    LOCAL PROC Path_Draw()
        MoveL point_0_clearance,v500,fine,GS25_ParallelGripper\WObj:=Workobject_1;
        MoveL point_0_contact,v500,fine,GS25_ParallelGripper\WObj:=Workobject_1;
        MoveL point_1_contact,v500,fine,GS25_ParallelGripper\WObj:=Workobject_1;
        MoveL point_1_clearance,v500,fine,GS25_ParallelGripper\WObj:=Workobject_1;
        MoveL point_2_clearance,v500,fine,GS25_ParallelGripper\WObj:=Workobject_1;
        MoveL point_2_contact,v500,fine,GS25_ParallelGripper\WObj:=Workobject_1;
        MoveL point_3_contact,v500,fine,GS25_ParallelGripper\WObj:=Workobject_1;
        MoveL point_3_clearance,v500,fine,GS25_ParallelGripper\WObj:=Workobject_1;
        MoveL point_4_clearance,v500,fine,GS25_ParallelGripper\WObj:=Workobject_1;
        MoveL point_4_contact,v500,fine,GS25_ParallelGripper\WObj:=Workobject_1;
        MoveL point_5_contact,v500,fine,GS25_ParallelGripper\WObj:=Workobject_1;
        MoveL point_5_clearance,v500,fine,GS25_ParallelGripper\WObj:=Workobject_1;
        MoveL point_6_clearance,v500,fine,GS25_ParallelGripper\WObj:=Workobject_1;
        MoveL point_6_contact,v500,fine,GS25_ParallelGripper\WObj:=Workobject_1;
        MoveL point_7_contact,v500,fine,GS25_ParallelGripper\WObj:=Workobject_1;
        MoveL point_7_clearance,v500,fine,GS25_ParallelGripper\WObj:=Workobject_1;
        MoveL point_8_clearance,v500,fine,GS25_ParallelGripper\WObj:=Workobject_1;
        MoveL point_8_contact,v500,fine,GS25_ParallelGripper\WObj:=Workobject_1;
        MoveL point_9_contact,v500,fine,GS25_ParallelGripper\WObj:=Workobject_1;
        MoveL point_9_clearance,v500,fine,GS25_ParallelGripper\WObj:=Workobject_1;
        MoveL point_10_clearance,v500,fine,GS25_ParallelGripper\WObj:=Workobject_1;
        MoveL point_10_contact,v500,fine,GS25_ParallelGripper\WObj:=Workobject_1;
        MoveL point_11_contact,v500,fine,GS25_ParallelGripper\WObj:=Workobject_1;
        MoveL point_11_clearance,v500,fine,GS25_ParallelGripper\WObj:=Workobject_1;
        MoveL point_12_clearance,v500,fine,GS25_ParallelGripper\WObj:=Workobject_1;
        MoveL point_12_contact,v500,fine,GS25_ParallelGripper\WObj:=Workobject_1;
        MoveL point_13_contact,v500,fine,GS25_ParallelGripper\WObj:=Workobject_1;
        MoveL point_13_clearance,v500,fine,GS25_ParallelGripper\WObj:=Workobject_1;
        MoveL point_14_clearance,v500,fine,GS25_ParallelGripper\WObj:=Workobject_1;
        MoveL point_14_contact,v500,fine,GS25_ParallelGripper\WObj:=Workobject_1;
        MoveL point_15_contact,v500,fine,GS25_ParallelGripper\WObj:=Workobject_1;
        MoveL point_15_clearance,v500,fine,GS25_ParallelGripper\WObj:=Workobject_1;
        MoveL point_16_clearance,v500,fine,GS25_ParallelGripper\WObj:=Workobject_1;
        MoveL point_16_contact,v500,fine,GS25_ParallelGripper\WObj:=Workobject_1;
        MoveL point_17_contact,v500,fine,GS25_ParallelGripper\WObj:=Workobject_1;
        MoveL point_17_clearance,v500,fine,GS25_ParallelGripper\WObj:=Workobject_1;
        MoveL point_18_clearance,v500,fine,GS25_ParallelGripper\WObj:=Workobject_1;
        MoveL point_18_contact,v500,fine,GS25_ParallelGripper\WObj:=Workobject_1;
        MoveL point_19_contact,v500,fine,GS25_ParallelGripper\WObj:=Workobject_1;
        MoveL point_19_clearance,v500,fine,GS25_ParallelGripper\WObj:=Workobject_1;
        MoveL point_20_clearance,v500,fine,GS25_ParallelGripper\WObj:=Workobject_1;
        MoveL point_20_contact,v500,fine,GS25_ParallelGripper\WObj:=Workobject_1;
        MoveL point_21_contact,v500,fine,GS25_ParallelGripper\WObj:=Workobject_1;
        MoveL point_21_clearance,v500,fine,GS25_ParallelGripper\WObj:=Workobject_1;
        MoveL point_22_clearance,v500,fine,GS25_ParallelGripper\WObj:=Workobject_1;
        MoveL point_22_contact,v500,fine,GS25_ParallelGripper\WObj:=Workobject_1;
        MoveL point_23_contact,v500,fine,GS25_ParallelGripper\WObj:=Workobject_1;
        MoveL point_23_clearance,v500,fine,GS25_ParallelGripper\WObj:=Workobject_1;
        MoveL point_24_clearance,v500,fine,GS25_ParallelGripper\WObj:=Workobject_1;
        MoveL point_24_contact,v500,fine,GS25_ParallelGripper\WObj:=Workobject_1;
        MoveL point_25_contact,v500,fine,GS25_ParallelGripper\WObj:=Workobject_1;
        MoveL point_25_clearance,v500,fine,GS25_ParallelGripper\WObj:=Workobject_1;
        MoveL point_26_clearance,v500,fine,GS25_ParallelGripper\WObj:=Workobject_1;
        MoveL point_26_contact,v500,fine,GS25_ParallelGripper\WObj:=Workobject_1;
        MoveL point_27_contact,v500,fine,GS25_ParallelGripper\WObj:=Workobject_1;
        MoveL point_27_clearance,v500,fine,GS25_ParallelGripper\WObj:=Workobject_1;
        MoveL point_28_clearance,v500,fine,GS25_ParallelGripper\WObj:=Workobject_1;
        MoveL point_28_contact,v500,fine,GS25_ParallelGripper\WObj:=Workobject_1;
        MoveL point_29_contact,v500,fine,GS25_ParallelGripper\WObj:=Workobject_1;
        MoveL point_29_clearance,v500,fine,GS25_ParallelGripper\WObj:=Workobject_1;
        MoveL point_30_clearance,v500,fine,GS25_ParallelGripper\WObj:=Workobject_1;
        MoveL point_30_contact,v500,fine,GS25_ParallelGripper\WObj:=Workobject_1;
        MoveL point_31_contact,v500,fine,GS25_ParallelGripper\WObj:=Workobject_1;
        MoveL point_31_clearance,v500,fine,GS25_ParallelGripper\WObj:=Workobject_1;
        MoveL point_32_clearance,v500,fine,GS25_ParallelGripper\WObj:=Workobject_1;
        MoveL point_32_contact,v500,fine,GS25_ParallelGripper\WObj:=Workobject_1;
        MoveL point_33_contact,v500,fine,GS25_ParallelGripper\WObj:=Workobject_1;
        MoveL point_33_clearance,v500,fine,GS25_ParallelGripper\WObj:=Workobject_1;
        MoveL point_34_clearance,v500,fine,GS25_ParallelGripper\WObj:=Workobject_1;
        MoveL point_34_contact,v500,fine,GS25_ParallelGripper\WObj:=Workobject_1;
        MoveL point_35_contact,v500,fine,GS25_ParallelGripper\WObj:=Workobject_1;
        MoveL point_35_clearance,v500,fine,GS25_ParallelGripper\WObj:=Workobject_1;
        MoveL point_36_clearance,v500,fine,GS25_ParallelGripper\WObj:=Workobject_1;
        MoveL point_36_contact,v500,fine,GS25_ParallelGripper\WObj:=Workobject_1;
        MoveL point_37_contact,v500,fine,GS25_ParallelGripper\WObj:=Workobject_1;
        MoveL point_37_clearance,v500,fine,GS25_ParallelGripper\WObj:=Workobject_1;
        MoveL point_38_clearance,v500,fine,GS25_ParallelGripper\WObj:=Workobject_1;
        MoveL point_38_contact,v500,fine,GS25_ParallelGripper\WObj:=Workobject_1;
        MoveL point_39_contact,v500,fine,GS25_ParallelGripper\WObj:=Workobject_1;
        MoveL point_39_clearance,v500,fine,GS25_ParallelGripper\WObj:=Workobject_1;
        MoveL point_40_clearance,v500,fine,GS25_ParallelGripper\WObj:=Workobject_1;
        MoveL point_40_contact,v500,fine,GS25_ParallelGripper\WObj:=Workobject_1;
        MoveL point_41_contact,v500,fine,GS25_ParallelGripper\WObj:=Workobject_1;
        MoveL point_41_clearance,v500,fine,GS25_ParallelGripper\WObj:=Workobject_1;
        MoveL point_42_clearance,v500,fine,GS25_ParallelGripper\WObj:=Workobject_1;
        MoveL point_42_contact,v500,fine,GS25_ParallelGripper\WObj:=Workobject_1;
        MoveL point_43_contact,v500,fine,GS25_ParallelGripper\WObj:=Workobject_1;
        MoveL point_43_clearance,v500,fine,GS25_ParallelGripper\WObj:=Workobject_1;
        MoveL point_44_clearance,v500,fine,GS25_ParallelGripper\WObj:=Workobject_1;
        MoveL point_44_contact,v500,fine,GS25_ParallelGripper\WObj:=Workobject_1;
        MoveL point_45_contact,v500,fine,GS25_ParallelGripper\WObj:=Workobject_1;
        MoveL point_45_clearance,v500,fine,GS25_ParallelGripper\WObj:=Workobject_1;
        MoveL point_46_clearance,v500,fine,GS25_ParallelGripper\WObj:=Workobject_1;
        MoveL point_46_contact,v500,fine,GS25_ParallelGripper\WObj:=Workobject_1;
        MoveL point_47_contact,v500,fine,GS25_ParallelGripper\WObj:=Workobject_1;
        MoveL point_47_clearance,v500,fine,GS25_ParallelGripper\WObj:=Workobject_1;
        MoveL point_48_clearance,v500,fine,GS25_ParallelGripper\WObj:=Workobject_1;
        MoveL point_48_contact,v500,fine,GS25_ParallelGripper\WObj:=Workobject_1;
        MoveL point_49_contact,v500,fine,GS25_ParallelGripper\WObj:=Workobject_1;
        MoveL point_49_clearance,v500,fine,GS25_ParallelGripper\WObj:=Workobject_1;
        MoveL point_50_clearance,v500,fine,GS25_ParallelGripper\WObj:=Workobject_1;
        MoveL point_50_contact,v500,fine,GS25_ParallelGripper\WObj:=Workobject_1;
        MoveL point_51_contact,v500,fine,GS25_ParallelGripper\WObj:=Workobject_1;
        MoveL point_51_clearance,v500,fine,GS25_ParallelGripper\WObj:=Workobject_1;
        MoveL point_52_clearance,v500,fine,GS25_ParallelGripper\WObj:=Workobject_1;
        MoveL point_52_contact,v500,fine,GS25_ParallelGripper\WObj:=Workobject_1;
        MoveL point_53_contact,v500,fine,GS25_ParallelGripper\WObj:=Workobject_1;
        MoveL point_53_clearance,v500,fine,GS25_ParallelGripper\WObj:=Workobject_1;
        MoveL point_54_clearance,v500,fine,GS25_ParallelGripper\WObj:=Workobject_1;
        MoveL point_54_contact,v500,fine,GS25_ParallelGripper\WObj:=Workobject_1;
        MoveL point_55_contact,v500,fine,GS25_ParallelGripper\WObj:=Workobject_1;
        MoveL point_55_clearance,v500,fine,GS25_ParallelGripper\WObj:=Workobject_1;
        MoveL point_56_clearance,v500,fine,GS25_ParallelGripper\WObj:=Workobject_1;
        MoveL point_56_contact,v500,fine,GS25_ParallelGripper\WObj:=Workobject_1;
        MoveL point_57_contact,v500,fine,GS25_ParallelGripper\WObj:=Workobject_1;
        MoveL point_57_clearance,v500,fine,GS25_ParallelGripper\WObj:=Workobject_1;
        MoveL point_58_clearance,v500,fine,GS25_ParallelGripper\WObj:=Workobject_1;
        MoveL point_58_contact,v500,fine,GS25_ParallelGripper\WObj:=Workobject_1;
        MoveL point_59_contact,v500,fine,GS25_ParallelGripper\WObj:=Workobject_1;
        MoveL point_59_clearance,v500,fine,GS25_ParallelGripper\WObj:=Workobject_1;
        MoveL point_60_clearance,v500,fine,GS25_ParallelGripper\WObj:=Workobject_1;
        MoveL point_60_contact,v500,fine,GS25_ParallelGripper\WObj:=Workobject_1;
        MoveL point_61_contact,v500,fine,GS25_ParallelGripper\WObj:=Workobject_1;
        MoveL point_61_clearance,v500,fine,GS25_ParallelGripper\WObj:=Workobject_1;
        MoveL point_62_clearance,v500,fine,GS25_ParallelGripper\WObj:=Workobject_1;
        MoveL point_62_contact,v500,fine,GS25_ParallelGripper\WObj:=Workobject_1;
        MoveL point_63_contact,v500,fine,GS25_ParallelGripper\WObj:=Workobject_1;
        MoveL point_63_clearance,v500,fine,GS25_ParallelGripper\WObj:=Workobject_1;
        MoveL point_64_clearance,v500,fine,GS25_ParallelGripper\WObj:=Workobject_1;
        MoveL point_64_contact,v500,fine,GS25_ParallelGripper\WObj:=Workobject_1;
        MoveL point_65_contact,v500,fine,GS25_ParallelGripper\WObj:=Workobject_1;
        MoveL point_65_clearance,v500,fine,GS25_ParallelGripper\WObj:=Workobject_1;
        MoveL point_66_clearance,v500,fine,GS25_ParallelGripper\WObj:=Workobject_1;
        MoveL point_66_contact,v500,fine,GS25_ParallelGripper\WObj:=Workobject_1;
        MoveL point_67_contact,v500,fine,GS25_ParallelGripper\WObj:=Workobject_1;
        MoveL point_67_clearance,v500,fine,GS25_ParallelGripper\WObj:=Workobject_1;
        MoveL point_68_clearance,v500,fine,GS25_ParallelGripper\WObj:=Workobject_1;
        MoveL point_68_contact,v500,fine,GS25_ParallelGripper\WObj:=Workobject_1;
        MoveL point_69_contact,v500,fine,GS25_ParallelGripper\WObj:=Workobject_1;
        MoveL point_69_clearance,v500,fine,GS25_ParallelGripper\WObj:=Workobject_1;
        MoveL point_70_clearance,v500,fine,GS25_ParallelGripper\WObj:=Workobject_1;
        MoveL point_70_contact,v500,fine,GS25_ParallelGripper\WObj:=Workobject_1;
        MoveL point_71_contact,v500,fine,GS25_ParallelGripper\WObj:=Workobject_1;
        MoveL point_71_clearance,v500,fine,GS25_ParallelGripper\WObj:=Workobject_1;
        MoveL point_72_clearance,v500,fine,GS25_ParallelGripper\WObj:=Workobject_1;
        MoveL point_72_contact,v500,fine,GS25_ParallelGripper\WObj:=Workobject_1;
        MoveL point_73_contact,v500,fine,GS25_ParallelGripper\WObj:=Workobject_1;
        MoveL point_73_clearance,v500,fine,GS25_ParallelGripper\WObj:=Workobject_1;
        MoveL point_74_clearance,v500,fine,GS25_ParallelGripper\WObj:=Workobject_1;
        MoveL point_74_contact,v500,fine,GS25_ParallelGripper\WObj:=Workobject_1;
        MoveL point_75_contact,v500,fine,GS25_ParallelGripper\WObj:=Workobject_1;
        MoveL point_75_clearance,v500,fine,GS25_ParallelGripper\WObj:=Workobject_1;
        MoveL point_76_clearance,v500,fine,GS25_ParallelGripper\WObj:=Workobject_1;
        MoveL point_76_contact,v500,fine,GS25_ParallelGripper\WObj:=Workobject_1;
        MoveL point_77_contact,v500,fine,GS25_ParallelGripper\WObj:=Workobject_1;
        MoveL point_77_clearance,v500,fine,GS25_ParallelGripper\WObj:=Workobject_1;
        MoveL point_78_clearance,v500,fine,GS25_ParallelGripper\WObj:=Workobject_1;
        MoveL point_78_contact,v500,fine,GS25_ParallelGripper\WObj:=Workobject_1;
        MoveL point_79_contact,v500,fine,GS25_ParallelGripper\WObj:=Workobject_1;
        MoveL point_79_clearance,v500,fine,GS25_ParallelGripper\WObj:=Workobject_1;
        MoveL point_80_clearance,v500,fine,GS25_ParallelGripper\WObj:=Workobject_1;
        MoveL point_80_contact,v500,fine,GS25_ParallelGripper\WObj:=Workobject_1;
        MoveL point_81_contact,v500,fine,GS25_ParallelGripper\WObj:=Workobject_1;
        MoveL point_81_clearance,v500,fine,GS25_ParallelGripper\WObj:=Workobject_1;
        MoveL point_82_clearance,v500,fine,GS25_ParallelGripper\WObj:=Workobject_1;
        MoveL point_82_contact,v500,fine,GS25_ParallelGripper\WObj:=Workobject_1;
        MoveL point_83_contact,v500,fine,GS25_ParallelGripper\WObj:=Workobject_1;
        MoveL point_83_clearance,v500,fine,GS25_ParallelGripper\WObj:=Workobject_1;
        MoveL point_84_clearance,v500,fine,GS25_ParallelGripper\WObj:=Workobject_1;
        MoveL point_84_contact,v500,fine,GS25_ParallelGripper\WObj:=Workobject_1;
        MoveL point_85_contact,v500,fine,GS25_ParallelGripper\WObj:=Workobject_1;
        MoveL point_85_clearance,v500,fine,GS25_ParallelGripper\WObj:=Workobject_1;
        MoveL point_86_clearance,v500,fine,GS25_ParallelGripper\WObj:=Workobject_1;
        MoveL point_86_contact,v500,fine,GS25_ParallelGripper\WObj:=Workobject_1;
        MoveL point_87_contact,v500,fine,GS25_ParallelGripper\WObj:=Workobject_1;
        MoveL point_87_clearance,v500,fine,GS25_ParallelGripper\WObj:=Workobject_1;
        MoveL point_88_clearance,v500,fine,GS25_ParallelGripper\WObj:=Workobject_1;
        MoveL point_88_contact,v500,fine,GS25_ParallelGripper\WObj:=Workobject_1;
        MoveL point_89_contact,v500,fine,GS25_ParallelGripper\WObj:=Workobject_1;
        MoveL point_89_clearance,v500,fine,GS25_ParallelGripper\WObj:=Workobject_1;
        MoveL point_90_clearance,v500,fine,GS25_ParallelGripper\WObj:=Workobject_1;
        MoveL point_90_contact,v500,fine,GS25_ParallelGripper\WObj:=Workobject_1;
        MoveL point_91_contact,v500,fine,GS25_ParallelGripper\WObj:=Workobject_1;
        MoveL point_91_clearance,v500,fine,GS25_ParallelGripper\WObj:=Workobject_1;
        MoveL point_92_clearance,v500,fine,GS25_ParallelGripper\WObj:=Workobject_1;
        MoveL point_92_contact,v500,fine,GS25_ParallelGripper\WObj:=Workobject_1;
        MoveL point_93_contact,v500,fine,GS25_ParallelGripper\WObj:=Workobject_1;
        MoveL point_93_clearance,v500,fine,GS25_ParallelGripper\WObj:=Workobject_1;
        MoveL point_94_clearance,v500,fine,GS25_ParallelGripper\WObj:=Workobject_1;
        MoveL point_94_contact,v500,fine,GS25_ParallelGripper\WObj:=Workobject_1;
        MoveL point_95_contact,v500,fine,GS25_ParallelGripper\WObj:=Workobject_1;
        MoveL point_95_clearance,v500,fine,GS25_ParallelGripper\WObj:=Workobject_1;
        MoveL point_96_clearance,v500,fine,GS25_ParallelGripper\WObj:=Workobject_1;
        MoveL point_96_contact,v500,fine,GS25_ParallelGripper\WObj:=Workobject_1;
        MoveL point_97_contact,v500,fine,GS25_ParallelGripper\WObj:=Workobject_1;
        MoveL point_97_clearance,v500,fine,GS25_ParallelGripper\WObj:=Workobject_1;
        MoveL point_98_clearance,v500,fine,GS25_ParallelGripper\WObj:=Workobject_1;
        MoveL point_98_contact,v500,fine,GS25_ParallelGripper\WObj:=Workobject_1;
        MoveL point_99_contact,v500,fine,GS25_ParallelGripper\WObj:=Workobject_1;
        MoveL point_99_clearance,v500,fine,GS25_ParallelGripper\WObj:=Workobject_1;
        MoveL point_100_clearance,v500,fine,GS25_ParallelGripper\WObj:=Workobject_1;
        MoveL point_100_contact,v500,fine,GS25_ParallelGripper\WObj:=Workobject_1;
        MoveL point_101_contact,v500,fine,GS25_ParallelGripper\WObj:=Workobject_1;
        MoveL point_101_clearance,v500,fine,GS25_ParallelGripper\WObj:=Workobject_1;
        MoveL point_102_clearance,v500,fine,GS25_ParallelGripper\WObj:=Workobject_1;
        MoveL point_102_contact,v500,fine,GS25_ParallelGripper\WObj:=Workobject_1;
        MoveL point_103_contact,v500,fine,GS25_ParallelGripper\WObj:=Workobject_1;
        MoveL point_103_clearance,v500,fine,GS25_ParallelGripper\WObj:=Workobject_1;
        MoveL point_104_clearance,v500,fine,GS25_ParallelGripper\WObj:=Workobject_1;
        MoveL point_104_contact,v500,fine,GS25_ParallelGripper\WObj:=Workobject_1;
        MoveL point_105_contact,v500,fine,GS25_ParallelGripper\WObj:=Workobject_1;
        MoveL point_105_clearance,v500,fine,GS25_ParallelGripper\WObj:=Workobject_1;
        MoveL point_106_clearance,v500,fine,GS25_ParallelGripper\WObj:=Workobject_1;
        MoveL point_106_contact,v500,fine,GS25_ParallelGripper\WObj:=Workobject_1;
        MoveL point_107_contact,v500,fine,GS25_ParallelGripper\WObj:=Workobject_1;
        MoveL point_107_clearance,v500,fine,GS25_ParallelGripper\WObj:=Workobject_1;
        MoveL point_108_clearance,v500,fine,GS25_ParallelGripper\WObj:=Workobject_1;
        MoveL point_108_contact,v500,fine,GS25_ParallelGripper\WObj:=Workobject_1;
        MoveL point_109_contact,v500,fine,GS25_ParallelGripper\WObj:=Workobject_1;
        MoveL point_109_clearance,v500,fine,GS25_ParallelGripper\WObj:=Workobject_1;
        MoveL point_110_clearance,v500,fine,GS25_ParallelGripper\WObj:=Workobject_1;
        MoveL point_110_contact,v500,fine,GS25_ParallelGripper\WObj:=Workobject_1;
        MoveL point_111_contact,v500,fine,GS25_ParallelGripper\WObj:=Workobject_1;
        MoveL point_111_clearance,v500,fine,GS25_ParallelGripper\WObj:=Workobject_1;
        MoveL point_112_clearance,v500,fine,GS25_ParallelGripper\WObj:=Workobject_1;
        MoveL point_112_contact,v500,fine,GS25_ParallelGripper\WObj:=Workobject_1;
        MoveL point_113_contact,v500,fine,GS25_ParallelGripper\WObj:=Workobject_1;
        MoveL point_113_clearance,v500,fine,GS25_ParallelGripper\WObj:=Workobject_1;
        MoveL point_114_clearance,v500,fine,GS25_ParallelGripper\WObj:=Workobject_1;
        MoveL point_114_contact,v500,fine,GS25_ParallelGripper\WObj:=Workobject_1;
        MoveL point_115_contact,v500,fine,GS25_ParallelGripper\WObj:=Workobject_1;
        MoveL point_115_clearance,v500,fine,GS25_ParallelGripper\WObj:=Workobject_1;
        MoveL point_116_clearance,v500,fine,GS25_ParallelGripper\WObj:=Workobject_1;
        MoveL point_116_contact,v500,fine,GS25_ParallelGripper\WObj:=Workobject_1;
        MoveL point_117_contact,v500,fine,GS25_ParallelGripper\WObj:=Workobject_1;
        MoveL point_117_clearance,v500,fine,GS25_ParallelGripper\WObj:=Workobject_1;
        MoveL point_118_clearance,v500,fine,GS25_ParallelGripper\WObj:=Workobject_1;
        MoveL point_118_contact,v500,fine,GS25_ParallelGripper\WObj:=Workobject_1;
        MoveL point_119_contact,v500,fine,GS25_ParallelGripper\WObj:=Workobject_1;
        MoveL point_119_clearance,v500,fine,GS25_ParallelGripper\WObj:=Workobject_1;
        MoveL point_120_clearance,v500,fine,GS25_ParallelGripper\WObj:=Workobject_1;
        MoveL point_120_contact,v500,fine,GS25_ParallelGripper\WObj:=Workobject_1;
        MoveL point_121_contact,v500,fine,GS25_ParallelGripper\WObj:=Workobject_1;
        MoveL point_121_clearance,v500,fine,GS25_ParallelGripper\WObj:=Workobject_1;
        MoveL point_122_clearance,v500,fine,GS25_ParallelGripper\WObj:=Workobject_1;
        MoveL point_122_contact,v500,fine,GS25_ParallelGripper\WObj:=Workobject_1;
        MoveL point_123_contact,v500,fine,GS25_ParallelGripper\WObj:=Workobject_1;
        MoveL point_123_clearance,v500,fine,GS25_ParallelGripper\WObj:=Workobject_1;
        MoveL point_124_clearance,v500,fine,GS25_ParallelGripper\WObj:=Workobject_1;
        MoveL point_124_contact,v500,fine,GS25_ParallelGripper\WObj:=Workobject_1;
        MoveL point_125_contact,v500,fine,GS25_ParallelGripper\WObj:=Workobject_1;
        MoveL point_125_clearance,v500,fine,GS25_ParallelGripper\WObj:=Workobject_1;
        MoveL point_126_clearance,v500,fine,GS25_ParallelGripper\WObj:=Workobject_1;
        MoveL point_126_contact,v500,fine,GS25_ParallelGripper\WObj:=Workobject_1;
        MoveL point_127_contact,v500,fine,GS25_ParallelGripper\WObj:=Workobject_1;
        MoveL point_127_clearance,v500,fine,GS25_ParallelGripper\WObj:=Workobject_1;
        MoveL point_128_clearance,v500,fine,GS25_ParallelGripper\WObj:=Workobject_1;
        MoveL point_128_contact,v500,fine,GS25_ParallelGripper\WObj:=Workobject_1;
        MoveL point_129_contact,v500,fine,GS25_ParallelGripper\WObj:=Workobject_1;
        MoveL point_129_clearance,v500,fine,GS25_ParallelGripper\WObj:=Workobject_1;
        MoveL point_130_clearance,v500,fine,GS25_ParallelGripper\WObj:=Workobject_1;
        MoveL point_130_contact,v500,fine,GS25_ParallelGripper\WObj:=Workobject_1;
        MoveL point_131_contact,v500,fine,GS25_ParallelGripper\WObj:=Workobject_1;
        MoveL point_131_clearance,v500,fine,GS25_ParallelGripper\WObj:=Workobject_1;
        MoveL point_132_clearance,v500,fine,GS25_ParallelGripper\WObj:=Workobject_1;
        MoveL point_132_contact,v500,fine,GS25_ParallelGripper\WObj:=Workobject_1;
        MoveL point_133_contact,v500,fine,GS25_ParallelGripper\WObj:=Workobject_1;
        MoveL point_133_clearance,v500,fine,GS25_ParallelGripper\WObj:=Workobject_1;
        MoveL point_134_clearance,v500,fine,GS25_ParallelGripper\WObj:=Workobject_1;
        MoveL point_134_contact,v500,fine,GS25_ParallelGripper\WObj:=Workobject_1;
        MoveL point_135_contact,v500,fine,GS25_ParallelGripper\WObj:=Workobject_1;
        MoveL point_135_clearance,v500,fine,GS25_ParallelGripper\WObj:=Workobject_1;
        MoveL point_136_clearance,v500,fine,GS25_ParallelGripper\WObj:=Workobject_1;
        MoveL point_136_contact,v500,fine,GS25_ParallelGripper\WObj:=Workobject_1;
        MoveL point_137_contact,v500,fine,GS25_ParallelGripper\WObj:=Workobject_1;
        MoveL point_137_clearance,v500,fine,GS25_ParallelGripper\WObj:=Workobject_1;
        MoveL point_138_clearance,v500,fine,GS25_ParallelGripper\WObj:=Workobject_1;
        MoveL point_138_contact,v500,fine,GS25_ParallelGripper\WObj:=Workobject_1;
        MoveL point_139_contact,v500,fine,GS25_ParallelGripper\WObj:=Workobject_1;
        MoveL point_139_clearance,v500,fine,GS25_ParallelGripper\WObj:=Workobject_1;
        MoveL point_140_clearance,v500,fine,GS25_ParallelGripper\WObj:=Workobject_1;
        MoveL point_140_contact,v500,fine,GS25_ParallelGripper\WObj:=Workobject_1;
        MoveL point_141_contact,v500,fine,GS25_ParallelGripper\WObj:=Workobject_1;
        MoveL point_141_clearance,v500,fine,GS25_ParallelGripper\WObj:=Workobject_1;
        MoveL point_142_clearance,v500,fine,GS25_ParallelGripper\WObj:=Workobject_1;
        MoveL point_142_contact,v500,fine,GS25_ParallelGripper\WObj:=Workobject_1;
        MoveL point_143_contact,v500,fine,GS25_ParallelGripper\WObj:=Workobject_1;
        MoveL point_143_clearance,v500,fine,GS25_ParallelGripper\WObj:=Workobject_1;
        MoveL point_144_clearance,v500,fine,GS25_ParallelGripper\WObj:=Workobject_1;
        MoveL point_144_contact,v500,fine,GS25_ParallelGripper\WObj:=Workobject_1;
        MoveL point_145_contact,v500,fine,GS25_ParallelGripper\WObj:=Workobject_1;
        MoveL point_145_clearance,v500,fine,GS25_ParallelGripper\WObj:=Workobject_1;
        MoveL point_146_clearance,v500,fine,GS25_ParallelGripper\WObj:=Workobject_1;
        MoveL point_146_contact,v500,fine,GS25_ParallelGripper\WObj:=Workobject_1;
        MoveL point_147_contact,v500,fine,GS25_ParallelGripper\WObj:=Workobject_1;
        MoveL point_147_clearance,v500,fine,GS25_ParallelGripper\WObj:=Workobject_1;
        MoveL point_148_clearance,v500,fine,GS25_ParallelGripper\WObj:=Workobject_1;
        MoveL point_148_contact,v500,fine,GS25_ParallelGripper\WObj:=Workobject_1;
        MoveL point_149_contact,v500,fine,GS25_ParallelGripper\WObj:=Workobject_1;
        MoveL point_149_clearance,v500,fine,GS25_ParallelGripper\WObj:=Workobject_1;
        MoveL point_150_clearance,v500,fine,GS25_ParallelGripper\WObj:=Workobject_1;
        MoveL point_150_contact,v500,fine,GS25_ParallelGripper\WObj:=Workobject_1;
        MoveL point_151_contact,v500,fine,GS25_ParallelGripper\WObj:=Workobject_1;
        MoveL point_151_clearance,v500,fine,GS25_ParallelGripper\WObj:=Workobject_1;
        MoveL point_152_clearance,v500,fine,GS25_ParallelGripper\WObj:=Workobject_1;
        MoveL point_152_contact,v500,fine,GS25_ParallelGripper\WObj:=Workobject_1;
        MoveL point_153_contact,v500,fine,GS25_ParallelGripper\WObj:=Workobject_1;
        MoveL point_153_clearance,v500,fine,GS25_ParallelGripper\WObj:=Workobject_1;
        MoveL point_154_clearance,v500,fine,GS25_ParallelGripper\WObj:=Workobject_1;
        MoveL point_154_contact,v500,fine,GS25_ParallelGripper\WObj:=Workobject_1;
        MoveL point_155_contact,v500,fine,GS25_ParallelGripper\WObj:=Workobject_1;
        MoveL point_155_clearance,v500,fine,GS25_ParallelGripper\WObj:=Workobject_1;
        MoveL point_156_clearance,v500,fine,GS25_ParallelGripper\WObj:=Workobject_1;
        MoveL point_156_contact,v500,fine,GS25_ParallelGripper\WObj:=Workobject_1;
        MoveL point_157_contact,v500,fine,GS25_ParallelGripper\WObj:=Workobject_1;
        MoveL point_157_clearance,v500,fine,GS25_ParallelGripper\WObj:=Workobject_1;
        MoveL point_158_clearance,v500,fine,GS25_ParallelGripper\WObj:=Workobject_1;
        MoveL point_158_contact,v500,fine,GS25_ParallelGripper\WObj:=Workobject_1;
        MoveL point_159_contact,v500,fine,GS25_ParallelGripper\WObj:=Workobject_1;
        MoveL point_159_clearance,v500,fine,GS25_ParallelGripper\WObj:=Workobject_1;
        MoveL point_160_clearance,v500,fine,GS25_ParallelGripper\WObj:=Workobject_1;
        MoveL point_160_contact,v500,fine,GS25_ParallelGripper\WObj:=Workobject_1;
        MoveL point_161_contact,v500,fine,GS25_ParallelGripper\WObj:=Workobject_1;
        MoveL point_161_clearance,v500,fine,GS25_ParallelGripper\WObj:=Workobject_1;
        MoveL point_162_clearance,v500,fine,GS25_ParallelGripper\WObj:=Workobject_1;
        MoveL point_162_contact,v500,fine,GS25_ParallelGripper\WObj:=Workobject_1;
        MoveL point_163_contact,v500,fine,GS25_ParallelGripper\WObj:=Workobject_1;
        MoveL point_163_clearance,v500,fine,GS25_ParallelGripper\WObj:=Workobject_1;
        MoveL point_164_clearance,v500,fine,GS25_ParallelGripper\WObj:=Workobject_1;
        MoveL point_164_contact,v500,fine,GS25_ParallelGripper\WObj:=Workobject_1;
        MoveL point_165_contact,v500,fine,GS25_ParallelGripper\WObj:=Workobject_1;
        MoveL point_165_clearance,v500,fine,GS25_ParallelGripper\WObj:=Workobject_1;
        MoveL point_166_clearance,v500,fine,GS25_ParallelGripper\WObj:=Workobject_1;
        MoveL point_166_contact,v500,fine,GS25_ParallelGripper\WObj:=Workobject_1;
        MoveL point_167_contact,v500,fine,GS25_ParallelGripper\WObj:=Workobject_1;
        MoveL point_167_clearance,v500,fine,GS25_ParallelGripper\WObj:=Workobject_1;
        MoveL point_168_clearance,v500,fine,GS25_ParallelGripper\WObj:=Workobject_1;
        MoveL point_168_contact,v500,fine,GS25_ParallelGripper\WObj:=Workobject_1;
        MoveL point_169_contact,v500,fine,GS25_ParallelGripper\WObj:=Workobject_1;
        MoveL point_169_clearance,v500,fine,GS25_ParallelGripper\WObj:=Workobject_1;
        MoveL point_170_clearance,v500,fine,GS25_ParallelGripper\WObj:=Workobject_1;
        MoveL point_170_contact,v500,fine,GS25_ParallelGripper\WObj:=Workobject_1;
        MoveL point_171_contact,v500,fine,GS25_ParallelGripper\WObj:=Workobject_1;
        MoveL point_171_clearance,v500,fine,GS25_ParallelGripper\WObj:=Workobject_1;
        MoveL point_172_clearance,v500,fine,GS25_ParallelGripper\WObj:=Workobject_1;
        MoveL point_172_contact,v500,fine,GS25_ParallelGripper\WObj:=Workobject_1;
        MoveL point_173_contact,v500,fine,GS25_ParallelGripper\WObj:=Workobject_1;
        MoveL point_173_clearance,v500,fine,GS25_ParallelGripper\WObj:=Workobject_1;
        MoveL point_174_clearance,v500,fine,GS25_ParallelGripper\WObj:=Workobject_1;
        MoveL point_174_contact,v500,fine,GS25_ParallelGripper\WObj:=Workobject_1;
        MoveL point_175_contact,v500,fine,GS25_ParallelGripper\WObj:=Workobject_1;
        MoveL point_175_clearance,v500,fine,GS25_ParallelGripper\WObj:=Workobject_1;
        MoveL point_176_clearance,v500,fine,GS25_ParallelGripper\WObj:=Workobject_1;
        MoveL point_176_contact,v500,fine,GS25_ParallelGripper\WObj:=Workobject_1;
        MoveL point_177_contact,v500,fine,GS25_ParallelGripper\WObj:=Workobject_1;
        MoveL point_177_clearance,v500,fine,GS25_ParallelGripper\WObj:=Workobject_1;
        MoveL point_178_clearance,v500,fine,GS25_ParallelGripper\WObj:=Workobject_1;
        MoveL point_178_contact,v500,fine,GS25_ParallelGripper\WObj:=Workobject_1;
        MoveL point_179_contact,v500,fine,GS25_ParallelGripper\WObj:=Workobject_1;
        MoveL point_179_clearance,v500,fine,GS25_ParallelGripper\WObj:=Workobject_1;
        MoveL point_180_clearance,v500,fine,GS25_ParallelGripper\WObj:=Workobject_1;
        MoveL point_180_contact,v500,fine,GS25_ParallelGripper\WObj:=Workobject_1;
        MoveL point_181_contact,v500,fine,GS25_ParallelGripper\WObj:=Workobject_1;
        MoveL point_181_clearance,v500,fine,GS25_ParallelGripper\WObj:=Workobject_1;
        MoveL point_182_clearance,v500,fine,GS25_ParallelGripper\WObj:=Workobject_1;
        MoveL point_182_contact,v500,fine,GS25_ParallelGripper\WObj:=Workobject_1;
        MoveL point_183_contact,v500,fine,GS25_ParallelGripper\WObj:=Workobject_1;
        MoveL point_183_clearance,v500,fine,GS25_ParallelGripper\WObj:=Workobject_1;
        MoveL point_184_clearance,v500,fine,GS25_ParallelGripper\WObj:=Workobject_1;
        MoveL point_184_contact,v500,fine,GS25_ParallelGripper\WObj:=Workobject_1;
        MoveL point_185_contact,v500,fine,GS25_ParallelGripper\WObj:=Workobject_1;
        MoveL point_185_clearance,v500,fine,GS25_ParallelGripper\WObj:=Workobject_1;
        MoveL point_186_clearance,v500,fine,GS25_ParallelGripper\WObj:=Workobject_1;
        MoveL point_186_contact,v500,fine,GS25_ParallelGripper\WObj:=Workobject_1;
        MoveL point_187_contact,v500,fine,GS25_ParallelGripper\WObj:=Workobject_1;
        MoveL point_187_clearance,v500,fine,GS25_ParallelGripper\WObj:=Workobject_1;
        MoveL point_188_clearance,v500,fine,GS25_ParallelGripper\WObj:=Workobject_1;
        MoveL point_188_contact,v500,fine,GS25_ParallelGripper\WObj:=Workobject_1;
        MoveL point_189_contact,v500,fine,GS25_ParallelGripper\WObj:=Workobject_1;
        MoveL point_189_clearance,v500,fine,GS25_ParallelGripper\WObj:=Workobject_1;
        MoveL point_190_clearance,v500,fine,GS25_ParallelGripper\WObj:=Workobject_1;
        MoveL point_190_contact,v500,fine,GS25_ParallelGripper\WObj:=Workobject_1;
        MoveL point_191_contact,v500,fine,GS25_ParallelGripper\WObj:=Workobject_1;
        MoveL point_191_clearance,v500,fine,GS25_ParallelGripper\WObj:=Workobject_1;
        MoveL point_192_clearance,v500,fine,GS25_ParallelGripper\WObj:=Workobject_1;
        MoveL point_192_contact,v500,fine,GS25_ParallelGripper\WObj:=Workobject_1;
        MoveL point_193_contact,v500,fine,GS25_ParallelGripper\WObj:=Workobject_1;
        MoveL point_193_clearance,v500,fine,GS25_ParallelGripper\WObj:=Workobject_1;
        MoveL point_194_clearance,v500,fine,GS25_ParallelGripper\WObj:=Workobject_1;
        MoveL point_194_contact,v500,fine,GS25_ParallelGripper\WObj:=Workobject_1;
        MoveL point_195_contact,v500,fine,GS25_ParallelGripper\WObj:=Workobject_1;
        MoveL point_195_clearance,v500,fine,GS25_ParallelGripper\WObj:=Workobject_1;
        MoveL point_196_clearance,v500,fine,GS25_ParallelGripper\WObj:=Workobject_1;
        MoveL point_196_contact,v500,fine,GS25_ParallelGripper\WObj:=Workobject_1;
        MoveL point_197_contact,v500,fine,GS25_ParallelGripper\WObj:=Workobject_1;
        MoveL point_197_clearance,v500,fine,GS25_ParallelGripper\WObj:=Workobject_1;
        MoveL point_198_clearance,v500,fine,GS25_ParallelGripper\WObj:=Workobject_1;
        MoveL point_198_contact,v500,fine,GS25_ParallelGripper\WObj:=Workobject_1;
        MoveL point_199_contact,v500,fine,GS25_ParallelGripper\WObj:=Workobject_1;
        MoveL point_199_clearance,v500,fine,GS25_ParallelGripper\WObj:=Workobject_1;
        MoveL point_200_clearance,v500,fine,GS25_ParallelGripper\WObj:=Workobject_1;
        MoveL point_200_contact,v500,fine,GS25_ParallelGripper\WObj:=Workobject_1;
        MoveL point_201_contact,v500,fine,GS25_ParallelGripper\WObj:=Workobject_1;
        MoveL point_201_clearance,v500,fine,GS25_ParallelGripper\WObj:=Workobject_1;
        MoveL point_202_clearance,v500,fine,GS25_ParallelGripper\WObj:=Workobject_1;
        MoveL point_202_contact,v500,fine,GS25_ParallelGripper\WObj:=Workobject_1;
        MoveL point_203_contact,v500,fine,GS25_ParallelGripper\WObj:=Workobject_1;
        MoveL point_203_clearance,v500,fine,GS25_ParallelGripper\WObj:=Workobject_1;
        MoveL point_204_clearance,v500,fine,GS25_ParallelGripper\WObj:=Workobject_1;
        MoveL point_204_contact,v500,fine,GS25_ParallelGripper\WObj:=Workobject_1;
        MoveL point_205_contact,v500,fine,GS25_ParallelGripper\WObj:=Workobject_1;
        MoveL point_205_clearance,v500,fine,GS25_ParallelGripper\WObj:=Workobject_1;
        MoveL point_206_clearance,v500,fine,GS25_ParallelGripper\WObj:=Workobject_1;
        MoveL point_206_contact,v500,fine,GS25_ParallelGripper\WObj:=Workobject_1;
        MoveL point_207_contact,v500,fine,GS25_ParallelGripper\WObj:=Workobject_1;
        MoveL point_207_clearance,v500,fine,GS25_ParallelGripper\WObj:=Workobject_1;
        MoveL point_208_clearance,v500,fine,GS25_ParallelGripper\WObj:=Workobject_1;
        MoveL point_208_contact,v500,fine,GS25_ParallelGripper\WObj:=Workobject_1;
        MoveL point_209_contact,v500,fine,GS25_ParallelGripper\WObj:=Workobject_1;
        MoveL point_209_clearance,v500,fine,GS25_ParallelGripper\WObj:=Workobject_1;
        MoveL point_210_clearance,v500,fine,GS25_ParallelGripper\WObj:=Workobject_1;
        MoveL point_210_contact,v500,fine,GS25_ParallelGripper\WObj:=Workobject_1;
        MoveL point_211_contact,v500,fine,GS25_ParallelGripper\WObj:=Workobject_1;
        MoveL point_211_clearance,v500,fine,GS25_ParallelGripper\WObj:=Workobject_1;
        MoveL point_212_clearance,v500,fine,GS25_ParallelGripper\WObj:=Workobject_1;
        MoveL point_212_contact,v500,fine,GS25_ParallelGripper\WObj:=Workobject_1;
        MoveL point_213_contact,v500,fine,GS25_ParallelGripper\WObj:=Workobject_1;
        MoveL point_213_clearance,v500,fine,GS25_ParallelGripper\WObj:=Workobject_1;
        MoveL point_214_clearance,v500,fine,GS25_ParallelGripper\WObj:=Workobject_1;
        MoveL point_214_contact,v500,fine,GS25_ParallelGripper\WObj:=Workobject_1;
        MoveL point_215_contact,v500,fine,GS25_ParallelGripper\WObj:=Workobject_1;
        MoveL point_215_clearance,v500,fine,GS25_ParallelGripper\WObj:=Workobject_1;
        MoveL point_216_clearance,v500,fine,GS25_ParallelGripper\WObj:=Workobject_1;
        MoveL point_216_contact,v500,fine,GS25_ParallelGripper\WObj:=Workobject_1;
        MoveL point_217_contact,v500,fine,GS25_ParallelGripper\WObj:=Workobject_1;
        MoveL point_217_clearance,v500,fine,GS25_ParallelGripper\WObj:=Workobject_1;
        MoveL point_218_clearance,v500,fine,GS25_ParallelGripper\WObj:=Workobject_1;
        MoveL point_218_contact,v500,fine,GS25_ParallelGripper\WObj:=Workobject_1;
        MoveL point_219_contact,v500,fine,GS25_ParallelGripper\WObj:=Workobject_1;
        MoveL point_219_clearance,v500,fine,GS25_ParallelGripper\WObj:=Workobject_1;
        MoveL point_220_clearance,v500,fine,GS25_ParallelGripper\WObj:=Workobject_1;
        MoveL point_220_contact,v500,fine,GS25_ParallelGripper\WObj:=Workobject_1;
        MoveL point_221_contact,v500,fine,GS25_ParallelGripper\WObj:=Workobject_1;
        MoveL point_221_clearance,v500,fine,GS25_ParallelGripper\WObj:=Workobject_1;
        MoveL point_222_clearance,v500,fine,GS25_ParallelGripper\WObj:=Workobject_1;
        MoveL point_222_contact,v500,fine,GS25_ParallelGripper\WObj:=Workobject_1;
        MoveL point_223_contact,v500,fine,GS25_ParallelGripper\WObj:=Workobject_1;
        MoveL point_223_clearance,v500,fine,GS25_ParallelGripper\WObj:=Workobject_1;
        MoveL point_224_clearance,v500,fine,GS25_ParallelGripper\WObj:=Workobject_1;
        MoveL point_224_contact,v500,fine,GS25_ParallelGripper\WObj:=Workobject_1;
        MoveL point_225_contact,v500,fine,GS25_ParallelGripper\WObj:=Workobject_1;
        MoveL point_225_clearance,v500,fine,GS25_ParallelGripper\WObj:=Workobject_1;
        MoveL point_226_clearance,v500,fine,GS25_ParallelGripper\WObj:=Workobject_1;
        MoveL point_226_contact,v500,fine,GS25_ParallelGripper\WObj:=Workobject_1;
        MoveL point_227_contact,v500,fine,GS25_ParallelGripper\WObj:=Workobject_1;
        MoveL point_227_clearance,v500,fine,GS25_ParallelGripper\WObj:=Workobject_1;
        MoveL point_228_clearance,v500,fine,GS25_ParallelGripper\WObj:=Workobject_1;
        MoveL point_228_contact,v500,fine,GS25_ParallelGripper\WObj:=Workobject_1;
        MoveL point_229_contact,v500,fine,GS25_ParallelGripper\WObj:=Workobject_1;
        MoveL point_229_clearance,v500,fine,GS25_ParallelGripper\WObj:=Workobject_1;
        MoveL point_230_clearance,v500,fine,GS25_ParallelGripper\WObj:=Workobject_1;
        MoveL point_230_contact,v500,fine,GS25_ParallelGripper\WObj:=Workobject_1;
        MoveL point_231_contact,v500,fine,GS25_ParallelGripper\WObj:=Workobject_1;
        MoveL point_231_clearance,v500,fine,GS25_ParallelGripper\WObj:=Workobject_1;
        MoveL point_232_clearance,v500,fine,GS25_ParallelGripper\WObj:=Workobject_1;
        MoveL point_232_contact,v500,fine,GS25_ParallelGripper\WObj:=Workobject_1;
        MoveL point_233_contact,v500,fine,GS25_ParallelGripper\WObj:=Workobject_1;
        MoveL point_233_clearance,v500,fine,GS25_ParallelGripper\WObj:=Workobject_1;
        MoveL point_234_clearance,v500,fine,GS25_ParallelGripper\WObj:=Workobject_1;
        MoveL point_234_contact,v500,fine,GS25_ParallelGripper\WObj:=Workobject_1;
        MoveL point_235_contact,v500,fine,GS25_ParallelGripper\WObj:=Workobject_1;
        MoveL point_235_clearance,v500,fine,GS25_ParallelGripper\WObj:=Workobject_1;
        MoveL point_236_clearance,v500,fine,GS25_ParallelGripper\WObj:=Workobject_1;
        MoveL point_236_contact,v500,fine,GS25_ParallelGripper\WObj:=Workobject_1;
        MoveL point_237_contact,v500,fine,GS25_ParallelGripper\WObj:=Workobject_1;
        MoveL point_237_clearance,v500,fine,GS25_ParallelGripper\WObj:=Workobject_1;
        MoveL point_238_clearance,v500,fine,GS25_ParallelGripper\WObj:=Workobject_1;
        MoveL point_238_contact,v500,fine,GS25_ParallelGripper\WObj:=Workobject_1;
        MoveL point_239_contact,v500,fine,GS25_ParallelGripper\WObj:=Workobject_1;
        MoveL point_239_clearance,v500,fine,GS25_ParallelGripper\WObj:=Workobject_1;
        MoveL point_240_clearance,v500,fine,GS25_ParallelGripper\WObj:=Workobject_1;
        MoveL point_240_contact,v500,fine,GS25_ParallelGripper\WObj:=Workobject_1;
        MoveL point_241_contact,v500,fine,GS25_ParallelGripper\WObj:=Workobject_1;
        MoveL point_241_clearance,v500,fine,GS25_ParallelGripper\WObj:=Workobject_1;
        MoveL point_242_clearance,v500,fine,GS25_ParallelGripper\WObj:=Workobject_1;
        MoveL point_242_contact,v500,fine,GS25_ParallelGripper\WObj:=Workobject_1;
        MoveL point_243_contact,v500,fine,GS25_ParallelGripper\WObj:=Workobject_1;
        MoveL point_243_clearance,v500,fine,GS25_ParallelGripper\WObj:=Workobject_1;
        MoveL point_244_clearance,v500,fine,GS25_ParallelGripper\WObj:=Workobject_1;
        MoveL point_244_contact,v500,fine,GS25_ParallelGripper\WObj:=Workobject_1;
        MoveL point_245_contact,v500,fine,GS25_ParallelGripper\WObj:=Workobject_1;
        MoveL point_245_clearance,v500,fine,GS25_ParallelGripper\WObj:=Workobject_1;
        MoveL point_246_clearance,v500,fine,GS25_ParallelGripper\WObj:=Workobject_1;
        MoveL point_246_contact,v500,fine,GS25_ParallelGripper\WObj:=Workobject_1;
        MoveL point_247_contact,v500,fine,GS25_ParallelGripper\WObj:=Workobject_1;
        MoveL point_247_clearance,v500,fine,GS25_ParallelGripper\WObj:=Workobject_1;
        MoveL point_248_clearance,v500,fine,GS25_ParallelGripper\WObj:=Workobject_1;
        MoveL point_248_contact,v500,fine,GS25_ParallelGripper\WObj:=Workobject_1;
        MoveL point_249_contact,v500,fine,GS25_ParallelGripper\WObj:=Workobject_1;
        MoveL point_249_clearance,v500,fine,GS25_ParallelGripper\WObj:=Workobject_1;
        MoveL point_250_clearance,v500,fine,GS25_ParallelGripper\WObj:=Workobject_1;
        MoveL point_250_contact,v500,fine,GS25_ParallelGripper\WObj:=Workobject_1;
        MoveL point_251_contact,v500,fine,GS25_ParallelGripper\WObj:=Workobject_1;
        MoveL point_251_clearance,v500,fine,GS25_ParallelGripper\WObj:=Workobject_1;
        MoveL point_252_clearance,v500,fine,GS25_ParallelGripper\WObj:=Workobject_1;
        MoveL point_252_contact,v500,fine,GS25_ParallelGripper\WObj:=Workobject_1;
        MoveL point_253_contact,v500,fine,GS25_ParallelGripper\WObj:=Workobject_1;
        MoveL point_253_clearance,v500,fine,GS25_ParallelGripper\WObj:=Workobject_1;
        MoveL point_254_clearance,v500,fine,GS25_ParallelGripper\WObj:=Workobject_1;
        MoveL point_254_contact,v500,fine,GS25_ParallelGripper\WObj:=Workobject_1;
        MoveL point_255_contact,v500,fine,GS25_ParallelGripper\WObj:=Workobject_1;
        MoveL point_255_clearance,v500,fine,GS25_ParallelGripper\WObj:=Workobject_1;
        MoveL point_256_clearance,v500,fine,GS25_ParallelGripper\WObj:=Workobject_1;
        MoveL point_256_contact,v500,fine,GS25_ParallelGripper\WObj:=Workobject_1;
        MoveL point_257_contact,v500,fine,GS25_ParallelGripper\WObj:=Workobject_1;
        MoveL point_257_clearance,v500,fine,GS25_ParallelGripper\WObj:=Workobject_1;
        MoveL point_258_clearance,v500,fine,GS25_ParallelGripper\WObj:=Workobject_1;
        MoveL point_258_contact,v500,fine,GS25_ParallelGripper\WObj:=Workobject_1;
        MoveL point_259_contact,v500,fine,GS25_ParallelGripper\WObj:=Workobject_1;
        MoveL point_259_clearance,v500,fine,GS25_ParallelGripper\WObj:=Workobject_1;
        MoveL point_260_clearance,v500,fine,GS25_ParallelGripper\WObj:=Workobject_1;
        MoveL point_260_contact,v500,fine,GS25_ParallelGripper\WObj:=Workobject_1;
        MoveL point_261_contact,v500,fine,GS25_ParallelGripper\WObj:=Workobject_1;
        MoveL point_261_clearance,v500,fine,GS25_ParallelGripper\WObj:=Workobject_1;
        MoveL point_262_clearance,v500,fine,GS25_ParallelGripper\WObj:=Workobject_1;
        MoveL point_262_contact,v500,fine,GS25_ParallelGripper\WObj:=Workobject_1;
        MoveL point_263_contact,v500,fine,GS25_ParallelGripper\WObj:=Workobject_1;
        MoveL point_263_clearance,v500,fine,GS25_ParallelGripper\WObj:=Workobject_1;
        MoveL point_264_clearance,v500,fine,GS25_ParallelGripper\WObj:=Workobject_1;
        MoveL point_264_contact,v500,fine,GS25_ParallelGripper\WObj:=Workobject_1;
        MoveL point_265_contact,v500,fine,GS25_ParallelGripper\WObj:=Workobject_1;
        MoveL point_265_clearance,v500,fine,GS25_ParallelGripper\WObj:=Workobject_1;
        MoveL point_266_clearance,v500,fine,GS25_ParallelGripper\WObj:=Workobject_1;
        MoveL point_266_contact,v500,fine,GS25_ParallelGripper\WObj:=Workobject_1;
        MoveL point_267_contact,v500,fine,GS25_ParallelGripper\WObj:=Workobject_1;
        MoveL point_267_clearance,v500,fine,GS25_ParallelGripper\WObj:=Workobject_1;
        MoveL point_268_clearance,v500,fine,GS25_ParallelGripper\WObj:=Workobject_1;
        MoveL point_268_contact,v500,fine,GS25_ParallelGripper\WObj:=Workobject_1;
        MoveL point_269_contact,v500,fine,GS25_ParallelGripper\WObj:=Workobject_1;
        MoveL point_269_clearance,v500,fine,GS25_ParallelGripper\WObj:=Workobject_1;
        MoveL point_270_clearance,v500,fine,GS25_ParallelGripper\WObj:=Workobject_1;
        MoveL point_270_contact,v500,fine,GS25_ParallelGripper\WObj:=Workobject_1;
        MoveL point_271_contact,v500,fine,GS25_ParallelGripper\WObj:=Workobject_1;
        MoveL point_271_clearance,v500,fine,GS25_ParallelGripper\WObj:=Workobject_1;
        MoveL point_272_clearance,v500,fine,GS25_ParallelGripper\WObj:=Workobject_1;
        MoveL point_272_contact,v500,fine,GS25_ParallelGripper\WObj:=Workobject_1;
        MoveL point_273_contact,v500,fine,GS25_ParallelGripper\WObj:=Workobject_1;
        MoveL point_273_clearance,v500,fine,GS25_ParallelGripper\WObj:=Workobject_1;
        MoveL point_274_clearance,v500,fine,GS25_ParallelGripper\WObj:=Workobject_1;
        MoveL point_274_contact,v500,fine,GS25_ParallelGripper\WObj:=Workobject_1;
        MoveL point_275_contact,v500,fine,GS25_ParallelGripper\WObj:=Workobject_1;
        MoveL point_275_clearance,v500,fine,GS25_ParallelGripper\WObj:=Workobject_1;
        MoveL point_276_clearance,v500,fine,GS25_ParallelGripper\WObj:=Workobject_1;
        MoveL point_276_contact,v500,fine,GS25_ParallelGripper\WObj:=Workobject_1;
        MoveL point_277_contact,v500,fine,GS25_ParallelGripper\WObj:=Workobject_1;
        MoveL point_277_clearance,v500,fine,GS25_ParallelGripper\WObj:=Workobject_1;
        MoveL point_278_clearance,v500,fine,GS25_ParallelGripper\WObj:=Workobject_1;
        MoveL point_278_contact,v500,fine,GS25_ParallelGripper\WObj:=Workobject_1;
        MoveL point_279_contact,v500,fine,GS25_ParallelGripper\WObj:=Workobject_1;
        MoveL point_279_clearance,v500,fine,GS25_ParallelGripper\WObj:=Workobject_1;
        MoveL point_280_clearance,v500,fine,GS25_ParallelGripper\WObj:=Workobject_1;
        MoveL point_280_contact,v500,fine,GS25_ParallelGripper\WObj:=Workobject_1;
        MoveL point_281_contact,v500,fine,GS25_ParallelGripper\WObj:=Workobject_1;
        MoveL point_281_clearance,v500,fine,GS25_ParallelGripper\WObj:=Workobject_1;
        MoveL point_282_clearance,v500,fine,GS25_ParallelGripper\WObj:=Workobject_1;
        MoveL point_282_contact,v500,fine,GS25_ParallelGripper\WObj:=Workobject_1;
        MoveL point_283_contact,v500,fine,GS25_ParallelGripper\WObj:=Workobject_1;
        MoveL point_283_clearance,v500,fine,GS25_ParallelGripper\WObj:=Workobject_1;
        MoveL point_284_clearance,v500,fine,GS25_ParallelGripper\WObj:=Workobject_1;
        MoveL point_284_contact,v500,fine,GS25_ParallelGripper\WObj:=Workobject_1;
        MoveL point_285_contact,v500,fine,GS25_ParallelGripper\WObj:=Workobject_1;
        MoveL point_285_clearance,v500,fine,GS25_ParallelGripper\WObj:=Workobject_1;
        MoveL point_286_clearance,v500,fine,GS25_ParallelGripper\WObj:=Workobject_1;
        MoveL point_286_contact,v500,fine,GS25_ParallelGripper\WObj:=Workobject_1;
        MoveL point_287_contact,v500,fine,GS25_ParallelGripper\WObj:=Workobject_1;
        MoveL point_287_clearance,v500,fine,GS25_ParallelGripper\WObj:=Workobject_1;
        MoveL point_288_clearance,v500,fine,GS25_ParallelGripper\WObj:=Workobject_1;
        MoveL point_288_contact,v500,fine,GS25_ParallelGripper\WObj:=Workobject_1;
        MoveL point_289_contact,v500,fine,GS25_ParallelGripper\WObj:=Workobject_1;
        MoveL point_289_clearance,v500,fine,GS25_ParallelGripper\WObj:=Workobject_1;
        MoveL point_290_clearance,v500,fine,GS25_ParallelGripper\WObj:=Workobject_1;
        MoveL point_290_contact,v500,fine,GS25_ParallelGripper\WObj:=Workobject_1;
        MoveL point_291_contact,v500,fine,GS25_ParallelGripper\WObj:=Workobject_1;
        MoveL point_291_clearance,v500,fine,GS25_ParallelGripper\WObj:=Workobject_1;
        MoveL point_292_clearance,v500,fine,GS25_ParallelGripper\WObj:=Workobject_1;
        MoveL point_292_contact,v500,fine,GS25_ParallelGripper\WObj:=Workobject_1;
        MoveL point_293_contact,v500,fine,GS25_ParallelGripper\WObj:=Workobject_1;
        MoveL point_293_clearance,v500,fine,GS25_ParallelGripper\WObj:=Workobject_1;
        MoveL point_294_clearance,v500,fine,GS25_ParallelGripper\WObj:=Workobject_1;
        MoveL point_294_contact,v500,fine,GS25_ParallelGripper\WObj:=Workobject_1;
        MoveL point_295_contact,v500,fine,GS25_ParallelGripper\WObj:=Workobject_1;
        MoveL point_295_clearance,v500,fine,GS25_ParallelGripper\WObj:=Workobject_1;
        MoveL point_296_clearance,v500,fine,GS25_ParallelGripper\WObj:=Workobject_1;
        MoveL point_296_contact,v500,fine,GS25_ParallelGripper\WObj:=Workobject_1;
        MoveL point_297_contact,v500,fine,GS25_ParallelGripper\WObj:=Workobject_1;
        MoveL point_297_clearance,v500,fine,GS25_ParallelGripper\WObj:=Workobject_1;
        MoveL point_298_clearance,v500,fine,GS25_ParallelGripper\WObj:=Workobject_1;
        MoveL point_298_contact,v500,fine,GS25_ParallelGripper\WObj:=Workobject_1;
        MoveL point_299_contact,v500,fine,GS25_ParallelGripper\WObj:=Workobject_1;
        MoveL point_299_clearance,v500,fine,GS25_ParallelGripper\WObj:=Workobject_1;
        MoveL point_300_clearance,v500,fine,GS25_ParallelGripper\WObj:=Workobject_1;
        MoveL point_300_contact,v500,fine,GS25_ParallelGripper\WObj:=Workobject_1;
        MoveL point_301_contact,v500,fine,GS25_ParallelGripper\WObj:=Workobject_1;
        MoveL point_301_clearance,v500,fine,GS25_ParallelGripper\WObj:=Workobject_1;
        MoveL point_302_clearance,v500,fine,GS25_ParallelGripper\WObj:=Workobject_1;
        MoveL point_302_contact,v500,fine,GS25_ParallelGripper\WObj:=Workobject_1;
        MoveL point_303_contact,v500,fine,GS25_ParallelGripper\WObj:=Workobject_1;
        MoveL point_303_clearance,v500,fine,GS25_ParallelGripper\WObj:=Workobject_1;
        MoveL point_304_clearance,v500,fine,GS25_ParallelGripper\WObj:=Workobject_1;
        MoveL point_304_contact,v500,fine,GS25_ParallelGripper\WObj:=Workobject_1;
        MoveL point_305_contact,v500,fine,GS25_ParallelGripper\WObj:=Workobject_1;
        MoveL point_305_clearance,v500,fine,GS25_ParallelGripper\WObj:=Workobject_1;
        MoveL point_306_clearance,v500,fine,GS25_ParallelGripper\WObj:=Workobject_1;
        MoveL point_306_contact,v500,fine,GS25_ParallelGripper\WObj:=Workobject_1;
        MoveL point_307_contact,v500,fine,GS25_ParallelGripper\WObj:=Workobject_1;
        MoveL point_307_clearance,v500,fine,GS25_ParallelGripper\WObj:=Workobject_1;
        MoveL point_308_clearance,v500,fine,GS25_ParallelGripper\WObj:=Workobject_1;
        MoveL point_308_contact,v500,fine,GS25_ParallelGripper\WObj:=Workobject_1;
        MoveL point_309_contact,v500,fine,GS25_ParallelGripper\WObj:=Workobject_1;
        MoveL point_309_clearance,v500,fine,GS25_ParallelGripper\WObj:=Workobject_1;
        MoveL point_310_clearance,v500,fine,GS25_ParallelGripper\WObj:=Workobject_1;
        MoveL point_310_contact,v500,fine,GS25_ParallelGripper\WObj:=Workobject_1;
        MoveL point_311_contact,v500,fine,GS25_ParallelGripper\WObj:=Workobject_1;
        MoveL point_311_clearance,v500,fine,GS25_ParallelGripper\WObj:=Workobject_1;
        MoveL point_312_clearance,v500,fine,GS25_ParallelGripper\WObj:=Workobject_1;
        MoveL point_312_contact,v500,fine,GS25_ParallelGripper\WObj:=Workobject_1;
        MoveL point_313_contact,v500,fine,GS25_ParallelGripper\WObj:=Workobject_1;
        MoveL point_313_clearance,v500,fine,GS25_ParallelGripper\WObj:=Workobject_1;
        MoveL point_314_clearance,v500,fine,GS25_ParallelGripper\WObj:=Workobject_1;
        MoveL point_314_contact,v500,fine,GS25_ParallelGripper\WObj:=Workobject_1;
        MoveL point_315_contact,v500,fine,GS25_ParallelGripper\WObj:=Workobject_1;
        MoveL point_315_clearance,v500,fine,GS25_ParallelGripper\WObj:=Workobject_1;
        MoveL point_316_clearance,v500,fine,GS25_ParallelGripper\WObj:=Workobject_1;
        MoveL point_316_contact,v500,fine,GS25_ParallelGripper\WObj:=Workobject_1;
        MoveL point_317_contact,v500,fine,GS25_ParallelGripper\WObj:=Workobject_1;
        MoveL point_317_clearance,v500,fine,GS25_ParallelGripper\WObj:=Workobject_1;
        MoveL point_318_clearance,v500,fine,GS25_ParallelGripper\WObj:=Workobject_1;
        MoveL point_318_contact,v500,fine,GS25_ParallelGripper\WObj:=Workobject_1;
        MoveL point_319_contact,v500,fine,GS25_ParallelGripper\WObj:=Workobject_1;
        MoveL point_319_clearance,v500,fine,GS25_ParallelGripper\WObj:=Workobject_1;
        MoveL point_320_clearance,v500,fine,GS25_ParallelGripper\WObj:=Workobject_1;
        MoveL point_320_contact,v500,fine,GS25_ParallelGripper\WObj:=Workobject_1;
        MoveL point_321_contact,v500,fine,GS25_ParallelGripper\WObj:=Workobject_1;
        MoveL point_321_clearance,v500,fine,GS25_ParallelGripper\WObj:=Workobject_1;
        MoveL point_322_clearance,v500,fine,GS25_ParallelGripper\WObj:=Workobject_1;
        MoveL point_322_contact,v500,fine,GS25_ParallelGripper\WObj:=Workobject_1;
        MoveL point_323_contact,v500,fine,GS25_ParallelGripper\WObj:=Workobject_1;
        MoveL point_323_clearance,v500,fine,GS25_ParallelGripper\WObj:=Workobject_1;
        MoveL point_324_clearance,v500,fine,GS25_ParallelGripper\WObj:=Workobject_1;
        MoveL point_324_contact,v500,fine,GS25_ParallelGripper\WObj:=Workobject_1;
        MoveL point_325_contact,v500,fine,GS25_ParallelGripper\WObj:=Workobject_1;
        MoveL point_325_clearance,v500,fine,GS25_ParallelGripper\WObj:=Workobject_1;
        MoveL point_326_clearance,v500,fine,GS25_ParallelGripper\WObj:=Workobject_1;
        MoveL point_326_contact,v500,fine,GS25_ParallelGripper\WObj:=Workobject_1;
        MoveL point_327_contact,v500,fine,GS25_ParallelGripper\WObj:=Workobject_1;
        MoveL point_327_clearance,v500,fine,GS25_ParallelGripper\WObj:=Workobject_1;
        MoveL point_328_clearance,v500,fine,GS25_ParallelGripper\WObj:=Workobject_1;
        MoveL point_328_contact,v500,fine,GS25_ParallelGripper\WObj:=Workobject_1;
        MoveL point_329_contact,v500,fine,GS25_ParallelGripper\WObj:=Workobject_1;
        MoveL point_329_clearance,v500,fine,GS25_ParallelGripper\WObj:=Workobject_1;
        MoveL point_330_clearance,v500,fine,GS25_ParallelGripper\WObj:=Workobject_1;
        MoveL point_330_contact,v500,fine,GS25_ParallelGripper\WObj:=Workobject_1;
        MoveL point_331_contact,v500,fine,GS25_ParallelGripper\WObj:=Workobject_1;
        MoveL point_331_clearance,v500,fine,GS25_ParallelGripper\WObj:=Workobject_1;
        MoveL point_332_clearance,v500,fine,GS25_ParallelGripper\WObj:=Workobject_1;
        MoveL point_332_contact,v500,fine,GS25_ParallelGripper\WObj:=Workobject_1;
        MoveL point_333_contact,v500,fine,GS25_ParallelGripper\WObj:=Workobject_1;
        MoveL point_333_clearance,v500,fine,GS25_ParallelGripper\WObj:=Workobject_1;
        MoveL point_334_clearance,v500,fine,GS25_ParallelGripper\WObj:=Workobject_1;
        MoveL point_334_contact,v500,fine,GS25_ParallelGripper\WObj:=Workobject_1;
        MoveL point_335_contact,v500,fine,GS25_ParallelGripper\WObj:=Workobject_1;
        MoveL point_335_clearance,v500,fine,GS25_ParallelGripper\WObj:=Workobject_1;
        MoveL point_336_clearance,v500,fine,GS25_ParallelGripper\WObj:=Workobject_1;
        MoveL point_336_contact,v500,fine,GS25_ParallelGripper\WObj:=Workobject_1;
        MoveL point_337_contact,v500,fine,GS25_ParallelGripper\WObj:=Workobject_1;
        MoveL point_337_clearance,v500,fine,GS25_ParallelGripper\WObj:=Workobject_1;
        MoveL point_338_clearance,v500,fine,GS25_ParallelGripper\WObj:=Workobject_1;
        MoveL point_338_contact,v500,fine,GS25_ParallelGripper\WObj:=Workobject_1;
        MoveL point_339_contact,v500,fine,GS25_ParallelGripper\WObj:=Workobject_1;
        MoveL point_339_clearance,v500,fine,GS25_ParallelGripper\WObj:=Workobject_1;
        MoveL point_340_clearance,v500,fine,GS25_ParallelGripper\WObj:=Workobject_1;
        MoveL point_340_contact,v500,fine,GS25_ParallelGripper\WObj:=Workobject_1;
        MoveL point_341_contact,v500,fine,GS25_ParallelGripper\WObj:=Workobject_1;
        MoveL point_341_clearance,v500,fine,GS25_ParallelGripper\WObj:=Workobject_1;
        MoveL point_342_clearance,v500,fine,GS25_ParallelGripper\WObj:=Workobject_1;
        MoveL point_342_contact,v500,fine,GS25_ParallelGripper\WObj:=Workobject_1;
        MoveL point_343_contact,v500,fine,GS25_ParallelGripper\WObj:=Workobject_1;
        MoveL point_343_clearance,v500,fine,GS25_ParallelGripper\WObj:=Workobject_1;
        MoveL point_344_clearance,v500,fine,GS25_ParallelGripper\WObj:=Workobject_1;
        MoveL point_344_contact,v500,fine,GS25_ParallelGripper\WObj:=Workobject_1;
        MoveL point_345_contact,v500,fine,GS25_ParallelGripper\WObj:=Workobject_1;
        MoveL point_345_clearance,v500,fine,GS25_ParallelGripper\WObj:=Workobject_1;
        MoveL point_346_clearance,v500,fine,GS25_ParallelGripper\WObj:=Workobject_1;
        MoveL point_346_contact,v500,fine,GS25_ParallelGripper\WObj:=Workobject_1;
        MoveL point_347_contact,v500,fine,GS25_ParallelGripper\WObj:=Workobject_1;
        MoveL point_347_clearance,v500,fine,GS25_ParallelGripper\WObj:=Workobject_1;
        MoveL point_348_clearance,v500,fine,GS25_ParallelGripper\WObj:=Workobject_1;
        MoveL point_348_contact,v500,fine,GS25_ParallelGripper\WObj:=Workobject_1;
        MoveL point_349_contact,v500,fine,GS25_ParallelGripper\WObj:=Workobject_1;
        MoveL point_349_clearance,v500,fine,GS25_ParallelGripper\WObj:=Workobject_1;
        MoveL point_350_clearance,v500,fine,GS25_ParallelGripper\WObj:=Workobject_1;
        MoveL point_350_contact,v500,fine,GS25_ParallelGripper\WObj:=Workobject_1;
        MoveL point_351_contact,v500,fine,GS25_ParallelGripper\WObj:=Workobject_1;
        MoveL point_351_clearance,v500,fine,GS25_ParallelGripper\WObj:=Workobject_1;
        MoveL point_352_clearance,v500,fine,GS25_ParallelGripper\WObj:=Workobject_1;
        MoveL point_352_contact,v500,fine,GS25_ParallelGripper\WObj:=Workobject_1;
        MoveL point_353_contact,v500,fine,GS25_ParallelGripper\WObj:=Workobject_1;
        MoveL point_353_clearance,v500,fine,GS25_ParallelGripper\WObj:=Workobject_1;
        MoveL point_354_clearance,v500,fine,GS25_ParallelGripper\WObj:=Workobject_1;
        MoveL point_354_contact,v500,fine,GS25_ParallelGripper\WObj:=Workobject_1;
        MoveL point_355_contact,v500,fine,GS25_ParallelGripper\WObj:=Workobject_1;
        MoveL point_355_clearance,v500,fine,GS25_ParallelGripper\WObj:=Workobject_1;
        MoveL point_356_clearance,v500,fine,GS25_ParallelGripper\WObj:=Workobject_1;
        MoveL point_356_contact,v500,fine,GS25_ParallelGripper\WObj:=Workobject_1;
        MoveL point_357_contact,v500,fine,GS25_ParallelGripper\WObj:=Workobject_1;
        MoveL point_357_clearance,v500,fine,GS25_ParallelGripper\WObj:=Workobject_1;
        MoveL point_358_clearance,v500,fine,GS25_ParallelGripper\WObj:=Workobject_1;
        MoveL point_358_contact,v500,fine,GS25_ParallelGripper\WObj:=Workobject_1;
        MoveL point_359_contact,v500,fine,GS25_ParallelGripper\WObj:=Workobject_1;
        MoveL point_359_clearance,v500,fine,GS25_ParallelGripper\WObj:=Workobject_1;
        MoveL point_360_clearance,v500,fine,GS25_ParallelGripper\WObj:=Workobject_1;
        MoveL point_360_contact,v500,fine,GS25_ParallelGripper\WObj:=Workobject_1;
        MoveL point_361_contact,v500,fine,GS25_ParallelGripper\WObj:=Workobject_1;
        MoveL point_361_clearance,v500,fine,GS25_ParallelGripper\WObj:=Workobject_1;
        MoveL point_362_clearance,v500,fine,GS25_ParallelGripper\WObj:=Workobject_1;
        MoveL point_362_contact,v500,fine,GS25_ParallelGripper\WObj:=Workobject_1;
        MoveL point_363_contact,v500,fine,GS25_ParallelGripper\WObj:=Workobject_1;
        MoveL point_363_clearance,v500,fine,GS25_ParallelGripper\WObj:=Workobject_1;
        MoveL point_364_clearance,v500,fine,GS25_ParallelGripper\WObj:=Workobject_1;
        MoveL point_364_contact,v500,fine,GS25_ParallelGripper\WObj:=Workobject_1;
        MoveL point_365_contact,v500,fine,GS25_ParallelGripper\WObj:=Workobject_1;
        MoveL point_365_clearance,v500,fine,GS25_ParallelGripper\WObj:=Workobject_1;
        MoveL point_366_clearance,v500,fine,GS25_ParallelGripper\WObj:=Workobject_1;
        MoveL point_366_contact,v500,fine,GS25_ParallelGripper\WObj:=Workobject_1;
        MoveL point_367_contact,v500,fine,GS25_ParallelGripper\WObj:=Workobject_1;
        MoveL point_367_clearance,v500,fine,GS25_ParallelGripper\WObj:=Workobject_1;
        MoveL point_368_clearance,v500,fine,GS25_ParallelGripper\WObj:=Workobject_1;
        MoveL point_368_contact,v500,fine,GS25_ParallelGripper\WObj:=Workobject_1;
        MoveL point_369_contact,v500,fine,GS25_ParallelGripper\WObj:=Workobject_1;
        MoveL point_369_clearance,v500,fine,GS25_ParallelGripper\WObj:=Workobject_1;
        MoveL point_370_clearance,v500,fine,GS25_ParallelGripper\WObj:=Workobject_1;
        MoveL point_370_contact,v500,fine,GS25_ParallelGripper\WObj:=Workobject_1;
        MoveL point_371_contact,v500,fine,GS25_ParallelGripper\WObj:=Workobject_1;
        MoveL point_371_clearance,v500,fine,GS25_ParallelGripper\WObj:=Workobject_1;
        MoveL point_372_clearance,v500,fine,GS25_ParallelGripper\WObj:=Workobject_1;
        MoveL point_372_contact,v500,fine,GS25_ParallelGripper\WObj:=Workobject_1;
        MoveL point_373_contact,v500,fine,GS25_ParallelGripper\WObj:=Workobject_1;
        MoveL point_373_clearance,v500,fine,GS25_ParallelGripper\WObj:=Workobject_1;
        MoveL point_374_clearance,v500,fine,GS25_ParallelGripper\WObj:=Workobject_1;
        MoveL point_374_contact,v500,fine,GS25_ParallelGripper\WObj:=Workobject_1;
        MoveL point_375_contact,v500,fine,GS25_ParallelGripper\WObj:=Workobject_1;
        MoveL point_375_clearance,v500,fine,GS25_ParallelGripper\WObj:=Workobject_1;
        MoveL point_376_clearance,v500,fine,GS25_ParallelGripper\WObj:=Workobject_1;
        MoveL point_376_contact,v500,fine,GS25_ParallelGripper\WObj:=Workobject_1;
        MoveL point_377_contact,v500,fine,GS25_ParallelGripper\WObj:=Workobject_1;
        MoveL point_377_clearance,v500,fine,GS25_ParallelGripper\WObj:=Workobject_1;
        MoveL point_378_clearance,v500,fine,GS25_ParallelGripper\WObj:=Workobject_1;
        MoveL point_378_contact,v500,fine,GS25_ParallelGripper\WObj:=Workobject_1;
        MoveL point_379_contact,v500,fine,GS25_ParallelGripper\WObj:=Workobject_1;
        MoveL point_379_clearance,v500,fine,GS25_ParallelGripper\WObj:=Workobject_1;
        MoveL point_380_clearance,v500,fine,GS25_ParallelGripper\WObj:=Workobject_1;
        MoveL point_380_contact,v500,fine,GS25_ParallelGripper\WObj:=Workobject_1;
        MoveL point_381_contact,v500,fine,GS25_ParallelGripper\WObj:=Workobject_1;
        MoveL point_381_clearance,v500,fine,GS25_ParallelGripper\WObj:=Workobject_1;
        MoveL point_382_clearance,v500,fine,GS25_ParallelGripper\WObj:=Workobject_1;
        MoveL point_382_contact,v500,fine,GS25_ParallelGripper\WObj:=Workobject_1;
        MoveL point_383_contact,v500,fine,GS25_ParallelGripper\WObj:=Workobject_1;
        MoveL point_383_clearance,v500,fine,GS25_ParallelGripper\WObj:=Workobject_1;
        MoveL point_384_clearance,v500,fine,GS25_ParallelGripper\WObj:=Workobject_1;
        MoveL point_384_contact,v500,fine,GS25_ParallelGripper\WObj:=Workobject_1;
        MoveL point_385_contact,v500,fine,GS25_ParallelGripper\WObj:=Workobject_1;
        MoveL point_385_clearance,v500,fine,GS25_ParallelGripper\WObj:=Workobject_1;
        MoveL point_386_clearance,v500,fine,GS25_ParallelGripper\WObj:=Workobject_1;
        MoveL point_386_contact,v500,fine,GS25_ParallelGripper\WObj:=Workobject_1;
        MoveL point_387_contact,v500,fine,GS25_ParallelGripper\WObj:=Workobject_1;
        MoveL point_387_clearance,v500,fine,GS25_ParallelGripper\WObj:=Workobject_1;
        MoveL point_388_clearance,v500,fine,GS25_ParallelGripper\WObj:=Workobject_1;
        MoveL point_388_contact,v500,fine,GS25_ParallelGripper\WObj:=Workobject_1;
        MoveL point_389_contact,v500,fine,GS25_ParallelGripper\WObj:=Workobject_1;
        MoveL point_389_clearance,v500,fine,GS25_ParallelGripper\WObj:=Workobject_1;
        MoveL point_390_clearance,v500,fine,GS25_ParallelGripper\WObj:=Workobject_1;
        MoveL point_390_contact,v500,fine,GS25_ParallelGripper\WObj:=Workobject_1;
        MoveL point_391_contact,v500,fine,GS25_ParallelGripper\WObj:=Workobject_1;
        MoveL point_391_clearance,v500,fine,GS25_ParallelGripper\WObj:=Workobject_1;
        MoveL point_392_clearance,v500,fine,GS25_ParallelGripper\WObj:=Workobject_1;
        MoveL point_392_contact,v500,fine,GS25_ParallelGripper\WObj:=Workobject_1;
        MoveL point_393_contact,v500,fine,GS25_ParallelGripper\WObj:=Workobject_1;
        MoveL point_393_clearance,v500,fine,GS25_ParallelGripper\WObj:=Workobject_1;
        MoveL point_394_clearance,v500,fine,GS25_ParallelGripper\WObj:=Workobject_1;
        MoveL point_394_contact,v500,fine,GS25_ParallelGripper\WObj:=Workobject_1;
        MoveL point_395_contact,v500,fine,GS25_ParallelGripper\WObj:=Workobject_1;
        MoveL point_395_clearance,v500,fine,GS25_ParallelGripper\WObj:=Workobject_1;
        MoveL point_396_clearance,v500,fine,GS25_ParallelGripper\WObj:=Workobject_1;
        MoveL point_396_contact,v500,fine,GS25_ParallelGripper\WObj:=Workobject_1;
        MoveL point_397_contact,v500,fine,GS25_ParallelGripper\WObj:=Workobject_1;
        MoveL point_397_clearance,v500,fine,GS25_ParallelGripper\WObj:=Workobject_1;
        MoveL point_398_clearance,v500,fine,GS25_ParallelGripper\WObj:=Workobject_1;
        MoveL point_398_contact,v500,fine,GS25_ParallelGripper\WObj:=Workobject_1;
        MoveL point_399_contact,v500,fine,GS25_ParallelGripper\WObj:=Workobject_1;
        MoveL point_399_clearance,v500,fine,GS25_ParallelGripper\WObj:=Workobject_1;
        MoveL point_400_clearance,v500,fine,GS25_ParallelGripper\WObj:=Workobject_1;
        MoveL point_400_contact,v500,fine,GS25_ParallelGripper\WObj:=Workobject_1;
        MoveL point_401_contact,v500,fine,GS25_ParallelGripper\WObj:=Workobject_1;
        MoveL point_401_clearance,v500,fine,GS25_ParallelGripper\WObj:=Workobject_1;
        MoveL point_402_clearance,v500,fine,GS25_ParallelGripper\WObj:=Workobject_1;
        MoveL point_402_contact,v500,fine,GS25_ParallelGripper\WObj:=Workobject_1;
        MoveL point_403_contact,v500,fine,GS25_ParallelGripper\WObj:=Workobject_1;
        MoveL point_403_clearance,v500,fine,GS25_ParallelGripper\WObj:=Workobject_1;
        MoveL point_404_clearance,v500,fine,GS25_ParallelGripper\WObj:=Workobject_1;
        MoveL point_404_contact,v500,fine,GS25_ParallelGripper\WObj:=Workobject_1;
        MoveL point_405_contact,v500,fine,GS25_ParallelGripper\WObj:=Workobject_1;
        MoveL point_405_clearance,v500,fine,GS25_ParallelGripper\WObj:=Workobject_1;
        MoveL point_406_clearance,v500,fine,GS25_ParallelGripper\WObj:=Workobject_1;
        MoveL point_406_contact,v500,fine,GS25_ParallelGripper\WObj:=Workobject_1;
        MoveL point_407_contact,v500,fine,GS25_ParallelGripper\WObj:=Workobject_1;
        MoveL point_407_clearance,v500,fine,GS25_ParallelGripper\WObj:=Workobject_1;
        MoveL point_408_clearance,v500,fine,GS25_ParallelGripper\WObj:=Workobject_1;
        MoveL point_408_contact,v500,fine,GS25_ParallelGripper\WObj:=Workobject_1;
        MoveL point_409_contact,v500,fine,GS25_ParallelGripper\WObj:=Workobject_1;
        MoveL point_409_clearance,v500,fine,GS25_ParallelGripper\WObj:=Workobject_1;
        MoveL point_410_clearance,v500,fine,GS25_ParallelGripper\WObj:=Workobject_1;
        MoveL point_410_contact,v500,fine,GS25_ParallelGripper\WObj:=Workobject_1;
        MoveL point_411_contact,v500,fine,GS25_ParallelGripper\WObj:=Workobject_1;
        MoveL point_411_clearance,v500,fine,GS25_ParallelGripper\WObj:=Workobject_1;
        MoveL point_412_clearance,v500,fine,GS25_ParallelGripper\WObj:=Workobject_1;
        MoveL point_412_contact,v500,fine,GS25_ParallelGripper\WObj:=Workobject_1;
        MoveL point_413_contact,v500,fine,GS25_ParallelGripper\WObj:=Workobject_1;
        MoveL point_413_clearance,v500,fine,GS25_ParallelGripper\WObj:=Workobject_1;
        MoveL point_414_clearance,v500,fine,GS25_ParallelGripper\WObj:=Workobject_1;
        MoveL point_414_contact,v500,fine,GS25_ParallelGripper\WObj:=Workobject_1;
        MoveL point_415_contact,v500,fine,GS25_ParallelGripper\WObj:=Workobject_1;
        MoveL point_415_clearance,v500,fine,GS25_ParallelGripper\WObj:=Workobject_1;
        MoveL point_416_clearance,v500,fine,GS25_ParallelGripper\WObj:=Workobject_1;
        MoveL point_416_contact,v500,fine,GS25_ParallelGripper\WObj:=Workobject_1;
        MoveL point_417_contact,v500,fine,GS25_ParallelGripper\WObj:=Workobject_1;
        MoveL point_417_clearance,v500,fine,GS25_ParallelGripper\WObj:=Workobject_1;
        MoveL point_418_clearance,v500,fine,GS25_ParallelGripper\WObj:=Workobject_1;
        MoveL point_418_contact,v500,fine,GS25_ParallelGripper\WObj:=Workobject_1;
        MoveL point_419_contact,v500,fine,GS25_ParallelGripper\WObj:=Workobject_1;
        MoveL point_419_clearance,v500,fine,GS25_ParallelGripper\WObj:=Workobject_1;
        MoveL point_420_clearance,v500,fine,GS25_ParallelGripper\WObj:=Workobject_1;
        MoveL point_420_contact,v500,fine,GS25_ParallelGripper\WObj:=Workobject_1;
        MoveL point_421_contact,v500,fine,GS25_ParallelGripper\WObj:=Workobject_1;
        MoveL point_421_clearance,v500,fine,GS25_ParallelGripper\WObj:=Workobject_1;
        MoveL point_422_clearance,v500,fine,GS25_ParallelGripper\WObj:=Workobject_1;
        MoveL point_422_contact,v500,fine,GS25_ParallelGripper\WObj:=Workobject_1;
        MoveL point_423_contact,v500,fine,GS25_ParallelGripper\WObj:=Workobject_1;
        MoveL point_423_clearance,v500,fine,GS25_ParallelGripper\WObj:=Workobject_1;
        MoveL point_424_clearance,v500,fine,GS25_ParallelGripper\WObj:=Workobject_1;
        MoveL point_424_contact,v500,fine,GS25_ParallelGripper\WObj:=Workobject_1;
        MoveL point_425_contact,v500,fine,GS25_ParallelGripper\WObj:=Workobject_1;
        MoveL point_425_clearance,v500,fine,GS25_ParallelGripper\WObj:=Workobject_1;
        MoveL point_426_clearance,v500,fine,GS25_ParallelGripper\WObj:=Workobject_1;
        MoveL point_426_contact,v500,fine,GS25_ParallelGripper\WObj:=Workobject_1;
        MoveL point_427_contact,v500,fine,GS25_ParallelGripper\WObj:=Workobject_1;
        MoveL point_427_clearance,v500,fine,GS25_ParallelGripper\WObj:=Workobject_1;
        MoveL point_428_clearance,v500,fine,GS25_ParallelGripper\WObj:=Workobject_1;
        MoveL point_428_contact,v500,fine,GS25_ParallelGripper\WObj:=Workobject_1;
        MoveL point_429_contact,v500,fine,GS25_ParallelGripper\WObj:=Workobject_1;
        MoveL point_429_clearance,v500,fine,GS25_ParallelGripper\WObj:=Workobject_1;
        MoveL point_430_clearance,v500,fine,GS25_ParallelGripper\WObj:=Workobject_1;
        MoveL point_430_contact,v500,fine,GS25_ParallelGripper\WObj:=Workobject_1;
        MoveL point_431_contact,v500,fine,GS25_ParallelGripper\WObj:=Workobject_1;
        MoveL point_431_clearance,v500,fine,GS25_ParallelGripper\WObj:=Workobject_1;
        MoveL point_432_clearance,v500,fine,GS25_ParallelGripper\WObj:=Workobject_1;
        MoveL point_432_contact,v500,fine,GS25_ParallelGripper\WObj:=Workobject_1;
        MoveL point_433_contact,v500,fine,GS25_ParallelGripper\WObj:=Workobject_1;
        MoveL point_433_clearance,v500,fine,GS25_ParallelGripper\WObj:=Workobject_1;
        MoveL point_434_clearance,v500,fine,GS25_ParallelGripper\WObj:=Workobject_1;
        MoveL point_434_contact,v500,fine,GS25_ParallelGripper\WObj:=Workobject_1;
        MoveL point_435_contact,v500,fine,GS25_ParallelGripper\WObj:=Workobject_1;
        MoveL point_435_clearance,v500,fine,GS25_ParallelGripper\WObj:=Workobject_1;
        MoveL point_436_clearance,v500,fine,GS25_ParallelGripper\WObj:=Workobject_1;
        MoveL point_436_contact,v500,fine,GS25_ParallelGripper\WObj:=Workobject_1;
        MoveL point_437_contact,v500,fine,GS25_ParallelGripper\WObj:=Workobject_1;
        MoveL point_437_clearance,v500,fine,GS25_ParallelGripper\WObj:=Workobject_1;
        MoveL point_438_clearance,v500,fine,GS25_ParallelGripper\WObj:=Workobject_1;
        MoveL point_438_contact,v500,fine,GS25_ParallelGripper\WObj:=Workobject_1;
        MoveL point_439_contact,v500,fine,GS25_ParallelGripper\WObj:=Workobject_1;
        MoveL point_439_clearance,v500,fine,GS25_ParallelGripper\WObj:=Workobject_1;
        MoveL point_440_clearance,v500,fine,GS25_ParallelGripper\WObj:=Workobject_1;
        MoveL point_440_contact,v500,fine,GS25_ParallelGripper\WObj:=Workobject_1;
        MoveL point_441_contact,v500,fine,GS25_ParallelGripper\WObj:=Workobject_1;
        MoveL point_441_clearance,v500,fine,GS25_ParallelGripper\WObj:=Workobject_1;
        MoveL point_442_clearance,v500,fine,GS25_ParallelGripper\WObj:=Workobject_1;
        MoveL point_442_contact,v500,fine,GS25_ParallelGripper\WObj:=Workobject_1;
        MoveL point_443_contact,v500,fine,GS25_ParallelGripper\WObj:=Workobject_1;
        MoveL point_443_clearance,v500,fine,GS25_ParallelGripper\WObj:=Workobject_1;
        MoveL point_444_clearance,v500,fine,GS25_ParallelGripper\WObj:=Workobject_1;
        MoveL point_444_contact,v500,fine,GS25_ParallelGripper\WObj:=Workobject_1;
        MoveL point_445_contact,v500,fine,GS25_ParallelGripper\WObj:=Workobject_1;
        MoveL point_445_clearance,v500,fine,GS25_ParallelGripper\WObj:=Workobject_1;
        MoveL point_446_clearance,v500,fine,GS25_ParallelGripper\WObj:=Workobject_1;
        MoveL point_446_contact,v500,fine,GS25_ParallelGripper\WObj:=Workobject_1;
        MoveL point_447_contact,v500,fine,GS25_ParallelGripper\WObj:=Workobject_1;
        MoveL point_447_clearance,v500,fine,GS25_ParallelGripper\WObj:=Workobject_1;
        MoveL point_448_clearance,v500,fine,GS25_ParallelGripper\WObj:=Workobject_1;
        MoveL point_448_contact,v500,fine,GS25_ParallelGripper\WObj:=Workobject_1;
        MoveL point_449_contact,v500,fine,GS25_ParallelGripper\WObj:=Workobject_1;
        MoveL point_449_clearance,v500,fine,GS25_ParallelGripper\WObj:=Workobject_1;
        MoveL point_450_clearance,v500,fine,GS25_ParallelGripper\WObj:=Workobject_1;
        MoveL point_450_contact,v500,fine,GS25_ParallelGripper\WObj:=Workobject_1;
        MoveL point_451_contact,v500,fine,GS25_ParallelGripper\WObj:=Workobject_1;
        MoveL point_451_clearance,v500,fine,GS25_ParallelGripper\WObj:=Workobject_1;
        MoveL point_452_clearance,v500,fine,GS25_ParallelGripper\WObj:=Workobject_1;
        MoveL point_452_contact,v500,fine,GS25_ParallelGripper\WObj:=Workobject_1;
        MoveL point_453_contact,v500,fine,GS25_ParallelGripper\WObj:=Workobject_1;
        MoveL point_453_clearance,v500,fine,GS25_ParallelGripper\WObj:=Workobject_1;
        MoveL point_454_clearance,v500,fine,GS25_ParallelGripper\WObj:=Workobject_1;
        MoveL point_454_contact,v500,fine,GS25_ParallelGripper\WObj:=Workobject_1;
        MoveL point_455_contact,v500,fine,GS25_ParallelGripper\WObj:=Workobject_1;
        MoveL point_455_clearance,v500,fine,GS25_ParallelGripper\WObj:=Workobject_1;
        MoveL point_456_clearance,v500,fine,GS25_ParallelGripper\WObj:=Workobject_1;
        MoveL point_456_contact,v500,fine,GS25_ParallelGripper\WObj:=Workobject_1;
        MoveL point_457_contact,v500,fine,GS25_ParallelGripper\WObj:=Workobject_1;
        MoveL point_457_clearance,v500,fine,GS25_ParallelGripper\WObj:=Workobject_1;
        MoveL point_458_clearance,v500,fine,GS25_ParallelGripper\WObj:=Workobject_1;
        MoveL point_458_contact,v500,fine,GS25_ParallelGripper\WObj:=Workobject_1;
        MoveL point_459_contact,v500,fine,GS25_ParallelGripper\WObj:=Workobject_1;
        MoveL point_459_clearance,v500,fine,GS25_ParallelGripper\WObj:=Workobject_1;
        MoveL point_460_clearance,v500,fine,GS25_ParallelGripper\WObj:=Workobject_1;
        MoveL point_460_contact,v500,fine,GS25_ParallelGripper\WObj:=Workobject_1;
        MoveL point_461_contact,v500,fine,GS25_ParallelGripper\WObj:=Workobject_1;
        MoveL point_461_clearance,v500,fine,GS25_ParallelGripper\WObj:=Workobject_1;
        MoveL point_462_clearance,v500,fine,GS25_ParallelGripper\WObj:=Workobject_1;
        MoveL point_462_contact,v500,fine,GS25_ParallelGripper\WObj:=Workobject_1;
        MoveL point_463_contact,v500,fine,GS25_ParallelGripper\WObj:=Workobject_1;
        MoveL point_463_clearance,v500,fine,GS25_ParallelGripper\WObj:=Workobject_1;
        MoveL point_464_clearance,v500,fine,GS25_ParallelGripper\WObj:=Workobject_1;
        MoveL point_464_contact,v500,fine,GS25_ParallelGripper\WObj:=Workobject_1;
        MoveL point_465_contact,v500,fine,GS25_ParallelGripper\WObj:=Workobject_1;
        MoveL point_465_clearance,v500,fine,GS25_ParallelGripper\WObj:=Workobject_1;
        MoveL point_466_clearance,v500,fine,GS25_ParallelGripper\WObj:=Workobject_1;
        MoveL point_466_contact,v500,fine,GS25_ParallelGripper\WObj:=Workobject_1;
        MoveL point_467_contact,v500,fine,GS25_ParallelGripper\WObj:=Workobject_1;
        MoveL point_467_clearance,v500,fine,GS25_ParallelGripper\WObj:=Workobject_1;
        MoveL point_468_clearance,v500,fine,GS25_ParallelGripper\WObj:=Workobject_1;
        MoveL point_468_contact,v500,fine,GS25_ParallelGripper\WObj:=Workobject_1;
        MoveL point_469_contact,v500,fine,GS25_ParallelGripper\WObj:=Workobject_1;
        MoveL point_469_clearance,v500,fine,GS25_ParallelGripper\WObj:=Workobject_1;
        MoveL point_470_clearance,v500,fine,GS25_ParallelGripper\WObj:=Workobject_1;
        MoveL point_470_contact,v500,fine,GS25_ParallelGripper\WObj:=Workobject_1;
        MoveL point_471_contact,v500,fine,GS25_ParallelGripper\WObj:=Workobject_1;
        MoveL point_471_clearance,v500,fine,GS25_ParallelGripper\WObj:=Workobject_1;
        MoveL point_472_clearance,v500,fine,GS25_ParallelGripper\WObj:=Workobject_1;
        MoveL point_472_contact,v500,fine,GS25_ParallelGripper\WObj:=Workobject_1;
        MoveL point_473_contact,v500,fine,GS25_ParallelGripper\WObj:=Workobject_1;
        MoveL point_473_clearance,v500,fine,GS25_ParallelGripper\WObj:=Workobject_1;
        MoveL point_474_clearance,v500,fine,GS25_ParallelGripper\WObj:=Workobject_1;
        MoveL point_474_contact,v500,fine,GS25_ParallelGripper\WObj:=Workobject_1;
        MoveL point_475_contact,v500,fine,GS25_ParallelGripper\WObj:=Workobject_1;
        MoveL point_475_clearance,v500,fine,GS25_ParallelGripper\WObj:=Workobject_1;
        MoveL point_476_clearance,v500,fine,GS25_ParallelGripper\WObj:=Workobject_1;
        MoveL point_476_contact,v500,fine,GS25_ParallelGripper\WObj:=Workobject_1;
        MoveL point_477_contact,v500,fine,GS25_ParallelGripper\WObj:=Workobject_1;
        MoveL point_477_clearance,v500,fine,GS25_ParallelGripper\WObj:=Workobject_1;
        MoveL point_478_clearance,v500,fine,GS25_ParallelGripper\WObj:=Workobject_1;
        MoveL point_478_contact,v500,fine,GS25_ParallelGripper\WObj:=Workobject_1;
        MoveL point_479_contact,v500,fine,GS25_ParallelGripper\WObj:=Workobject_1;
        MoveL point_479_clearance,v500,fine,GS25_ParallelGripper\WObj:=Workobject_1;
        MoveL point_480_clearance,v500,fine,GS25_ParallelGripper\WObj:=Workobject_1;
        MoveL point_480_contact,v500,fine,GS25_ParallelGripper\WObj:=Workobject_1;
        MoveL point_481_contact,v500,fine,GS25_ParallelGripper\WObj:=Workobject_1;
        MoveL point_481_clearance,v500,fine,GS25_ParallelGripper\WObj:=Workobject_1;
        MoveL point_482_clearance,v500,fine,GS25_ParallelGripper\WObj:=Workobject_1;
        MoveL point_482_contact,v500,fine,GS25_ParallelGripper\WObj:=Workobject_1;
        MoveL point_483_contact,v500,fine,GS25_ParallelGripper\WObj:=Workobject_1;
        MoveL point_483_clearance,v500,fine,GS25_ParallelGripper\WObj:=Workobject_1;
        MoveL point_484_clearance,v500,fine,GS25_ParallelGripper\WObj:=Workobject_1;
        MoveL point_484_contact,v500,fine,GS25_ParallelGripper\WObj:=Workobject_1;
        MoveL point_485_contact,v500,fine,GS25_ParallelGripper\WObj:=Workobject_1;
        MoveL point_485_clearance,v500,fine,GS25_ParallelGripper\WObj:=Workobject_1;
        MoveL point_486_clearance,v500,fine,GS25_ParallelGripper\WObj:=Workobject_1;
        MoveL point_486_contact,v500,fine,GS25_ParallelGripper\WObj:=Workobject_1;
        MoveL point_487_contact,v500,fine,GS25_ParallelGripper\WObj:=Workobject_1;
        MoveL point_487_clearance,v500,fine,GS25_ParallelGripper\WObj:=Workobject_1;
        MoveL point_488_clearance,v500,fine,GS25_ParallelGripper\WObj:=Workobject_1;
        MoveL point_488_contact,v500,fine,GS25_ParallelGripper\WObj:=Workobject_1;
        MoveL point_489_contact,v500,fine,GS25_ParallelGripper\WObj:=Workobject_1;
        MoveL point_489_clearance,v500,fine,GS25_ParallelGripper\WObj:=Workobject_1;
        MoveL point_490_clearance,v500,fine,GS25_ParallelGripper\WObj:=Workobject_1;
        MoveL point_490_contact,v500,fine,GS25_ParallelGripper\WObj:=Workobject_1;
        MoveL point_491_contact,v500,fine,GS25_ParallelGripper\WObj:=Workobject_1;
        MoveL point_491_clearance,v500,fine,GS25_ParallelGripper\WObj:=Workobject_1;
        MoveL point_492_clearance,v500,fine,GS25_ParallelGripper\WObj:=Workobject_1;
        MoveL point_492_contact,v500,fine,GS25_ParallelGripper\WObj:=Workobject_1;
        MoveL point_493_contact,v500,fine,GS25_ParallelGripper\WObj:=Workobject_1;
        MoveL point_493_clearance,v500,fine,GS25_ParallelGripper\WObj:=Workobject_1;
        MoveL point_494_clearance,v500,fine,GS25_ParallelGripper\WObj:=Workobject_1;
        MoveL point_494_contact,v500,fine,GS25_ParallelGripper\WObj:=Workobject_1;
        MoveL point_495_contact,v500,fine,GS25_ParallelGripper\WObj:=Workobject_1;
        MoveL point_495_clearance,v500,fine,GS25_ParallelGripper\WObj:=Workobject_1;
        MoveL point_496_clearance,v500,fine,GS25_ParallelGripper\WObj:=Workobject_1;
        MoveL point_496_contact,v500,fine,GS25_ParallelGripper\WObj:=Workobject_1;
        MoveL point_497_contact,v500,fine,GS25_ParallelGripper\WObj:=Workobject_1;
        MoveL point_497_clearance,v500,fine,GS25_ParallelGripper\WObj:=Workobject_1;
        MoveL point_498_clearance,v500,fine,GS25_ParallelGripper\WObj:=Workobject_1;
        MoveL point_498_contact,v500,fine,GS25_ParallelGripper\WObj:=Workobject_1;
        MoveL point_499_contact,v500,fine,GS25_ParallelGripper\WObj:=Workobject_1;
        MoveL point_499_clearance,v500,fine,GS25_ParallelGripper\WObj:=Workobject_1;
        MoveL point_500_clearance,v500,fine,GS25_ParallelGripper\WObj:=Workobject_1;
        MoveL point_500_contact,v500,fine,GS25_ParallelGripper\WObj:=Workobject_1;
        MoveL point_501_contact,v500,fine,GS25_ParallelGripper\WObj:=Workobject_1;
        MoveL point_501_clearance,v500,fine,GS25_ParallelGripper\WObj:=Workobject_1;
        MoveL point_502_clearance,v500,fine,GS25_ParallelGripper\WObj:=Workobject_1;
        MoveL point_502_contact,v500,fine,GS25_ParallelGripper\WObj:=Workobject_1;
        MoveL point_503_contact,v500,fine,GS25_ParallelGripper\WObj:=Workobject_1;
        MoveL point_503_clearance,v500,fine,GS25_ParallelGripper\WObj:=Workobject_1;
        MoveL point_504_clearance,v500,fine,GS25_ParallelGripper\WObj:=Workobject_1;
        MoveL point_504_contact,v500,fine,GS25_ParallelGripper\WObj:=Workobject_1;
        MoveL point_505_contact,v500,fine,GS25_ParallelGripper\WObj:=Workobject_1;
        MoveL point_505_clearance,v500,fine,GS25_ParallelGripper\WObj:=Workobject_1;
        MoveL point_506_clearance,v500,fine,GS25_ParallelGripper\WObj:=Workobject_1;
        MoveL point_506_contact,v500,fine,GS25_ParallelGripper\WObj:=Workobject_1;
        MoveL point_507_contact,v500,fine,GS25_ParallelGripper\WObj:=Workobject_1;
        MoveL point_507_clearance,v500,fine,GS25_ParallelGripper\WObj:=Workobject_1;
        MoveL point_508_clearance,v500,fine,GS25_ParallelGripper\WObj:=Workobject_1;
        MoveL point_508_contact,v500,fine,GS25_ParallelGripper\WObj:=Workobject_1;
        MoveL point_509_contact,v500,fine,GS25_ParallelGripper\WObj:=Workobject_1;
        MoveL point_509_clearance,v500,fine,GS25_ParallelGripper\WObj:=Workobject_1;
        MoveL point_510_clearance,v500,fine,GS25_ParallelGripper\WObj:=Workobject_1;
        MoveL point_510_contact,v500,fine,GS25_ParallelGripper\WObj:=Workobject_1;
        MoveL point_511_contact,v500,fine,GS25_ParallelGripper\WObj:=Workobject_1;
        MoveL point_511_clearance,v500,fine,GS25_ParallelGripper\WObj:=Workobject_1;
        MoveL point_512_clearance,v500,fine,GS25_ParallelGripper\WObj:=Workobject_1;
        MoveL point_512_contact,v500,fine,GS25_ParallelGripper\WObj:=Workobject_1;
        MoveL point_513_contact,v500,fine,GS25_ParallelGripper\WObj:=Workobject_1;
        MoveL point_513_clearance,v500,fine,GS25_ParallelGripper\WObj:=Workobject_1;
        MoveL point_514_clearance,v500,fine,GS25_ParallelGripper\WObj:=Workobject_1;
        MoveL point_514_contact,v500,fine,GS25_ParallelGripper\WObj:=Workobject_1;
        MoveL point_515_contact,v500,fine,GS25_ParallelGripper\WObj:=Workobject_1;
        MoveL point_515_clearance,v500,fine,GS25_ParallelGripper\WObj:=Workobject_1;
        MoveL point_516_clearance,v500,fine,GS25_ParallelGripper\WObj:=Workobject_1;
        MoveL point_516_contact,v500,fine,GS25_ParallelGripper\WObj:=Workobject_1;
        MoveL point_517_contact,v500,fine,GS25_ParallelGripper\WObj:=Workobject_1;
        MoveL point_517_clearance,v500,fine,GS25_ParallelGripper\WObj:=Workobject_1;
        MoveL point_518_clearance,v500,fine,GS25_ParallelGripper\WObj:=Workobject_1;
        MoveL point_518_contact,v500,fine,GS25_ParallelGripper\WObj:=Workobject_1;
        MoveL point_519_contact,v500,fine,GS25_ParallelGripper\WObj:=Workobject_1;
        MoveL point_519_clearance,v500,fine,GS25_ParallelGripper\WObj:=Workobject_1;
        MoveL point_520_clearance,v500,fine,GS25_ParallelGripper\WObj:=Workobject_1;
        MoveL point_520_contact,v500,fine,GS25_ParallelGripper\WObj:=Workobject_1;
        MoveL point_521_contact,v500,fine,GS25_ParallelGripper\WObj:=Workobject_1;
        MoveL point_521_clearance,v500,fine,GS25_ParallelGripper\WObj:=Workobject_1;
        MoveL point_522_clearance,v500,fine,GS25_ParallelGripper\WObj:=Workobject_1;
        MoveL point_522_contact,v500,fine,GS25_ParallelGripper\WObj:=Workobject_1;
        MoveL point_523_contact,v500,fine,GS25_ParallelGripper\WObj:=Workobject_1;
        MoveL point_523_clearance,v500,fine,GS25_ParallelGripper\WObj:=Workobject_1;
        MoveL point_524_clearance,v500,fine,GS25_ParallelGripper\WObj:=Workobject_1;
        MoveL point_524_contact,v500,fine,GS25_ParallelGripper\WObj:=Workobject_1;
        MoveL point_525_contact,v500,fine,GS25_ParallelGripper\WObj:=Workobject_1;
        MoveL point_525_clearance,v500,fine,GS25_ParallelGripper\WObj:=Workobject_1;
        MoveL point_526_clearance,v500,fine,GS25_ParallelGripper\WObj:=Workobject_1;
        MoveL point_526_contact,v500,fine,GS25_ParallelGripper\WObj:=Workobject_1;
        MoveL point_527_contact,v500,fine,GS25_ParallelGripper\WObj:=Workobject_1;
        MoveL point_527_clearance,v500,fine,GS25_ParallelGripper\WObj:=Workobject_1;
        MoveL point_528_clearance,v500,fine,GS25_ParallelGripper\WObj:=Workobject_1;
        MoveL point_528_contact,v500,fine,GS25_ParallelGripper\WObj:=Workobject_1;
        MoveL point_529_contact,v500,fine,GS25_ParallelGripper\WObj:=Workobject_1;
        MoveL point_529_clearance,v500,fine,GS25_ParallelGripper\WObj:=Workobject_1;
        MoveL point_530_clearance,v500,fine,GS25_ParallelGripper\WObj:=Workobject_1;
        MoveL point_530_contact,v500,fine,GS25_ParallelGripper\WObj:=Workobject_1;
        MoveL point_531_contact,v500,fine,GS25_ParallelGripper\WObj:=Workobject_1;
        MoveL point_531_clearance,v500,fine,GS25_ParallelGripper\WObj:=Workobject_1;
        MoveL point_532_clearance,v500,fine,GS25_ParallelGripper\WObj:=Workobject_1;
        MoveL point_532_contact,v500,fine,GS25_ParallelGripper\WObj:=Workobject_1;
        MoveL point_533_contact,v500,fine,GS25_ParallelGripper\WObj:=Workobject_1;
        MoveL point_533_clearance,v500,fine,GS25_ParallelGripper\WObj:=Workobject_1;
        MoveL point_534_clearance,v500,fine,GS25_ParallelGripper\WObj:=Workobject_1;
        MoveL point_534_contact,v500,fine,GS25_ParallelGripper\WObj:=Workobject_1;
        MoveL point_535_contact,v500,fine,GS25_ParallelGripper\WObj:=Workobject_1;
        MoveL point_535_clearance,v500,fine,GS25_ParallelGripper\WObj:=Workobject_1;
        MoveL point_536_clearance,v500,fine,GS25_ParallelGripper\WObj:=Workobject_1;
        MoveL point_536_contact,v500,fine,GS25_ParallelGripper\WObj:=Workobject_1;
        MoveL point_537_contact,v500,fine,GS25_ParallelGripper\WObj:=Workobject_1;
        MoveL point_537_clearance,v500,fine,GS25_ParallelGripper\WObj:=Workobject_1;
        MoveL point_538_clearance,v500,fine,GS25_ParallelGripper\WObj:=Workobject_1;
        MoveL point_538_contact,v500,fine,GS25_ParallelGripper\WObj:=Workobject_1;
        MoveL point_539_contact,v500,fine,GS25_ParallelGripper\WObj:=Workobject_1;
        MoveL point_539_clearance,v500,fine,GS25_ParallelGripper\WObj:=Workobject_1;
        MoveL point_540_clearance,v500,fine,GS25_ParallelGripper\WObj:=Workobject_1;
        MoveL point_540_contact,v500,fine,GS25_ParallelGripper\WObj:=Workobject_1;
        MoveL point_541_contact,v500,fine,GS25_ParallelGripper\WObj:=Workobject_1;
        MoveL point_541_clearance,v500,fine,GS25_ParallelGripper\WObj:=Workobject_1;
        MoveL point_542_clearance,v500,fine,GS25_ParallelGripper\WObj:=Workobject_1;
        MoveL point_542_contact,v500,fine,GS25_ParallelGripper\WObj:=Workobject_1;
        MoveL point_543_contact,v500,fine,GS25_ParallelGripper\WObj:=Workobject_1;
        MoveL point_543_clearance,v500,fine,GS25_ParallelGripper\WObj:=Workobject_1;
        MoveL point_544_clearance,v500,fine,GS25_ParallelGripper\WObj:=Workobject_1;
        MoveL point_544_contact,v500,fine,GS25_ParallelGripper\WObj:=Workobject_1;
        MoveL point_545_contact,v500,fine,GS25_ParallelGripper\WObj:=Workobject_1;
        MoveL point_545_clearance,v500,fine,GS25_ParallelGripper\WObj:=Workobject_1;
        MoveL point_546_clearance,v500,fine,GS25_ParallelGripper\WObj:=Workobject_1;
        MoveL point_546_contact,v500,fine,GS25_ParallelGripper\WObj:=Workobject_1;
        MoveL point_547_contact,v500,fine,GS25_ParallelGripper\WObj:=Workobject_1;
        MoveL point_547_clearance,v500,fine,GS25_ParallelGripper\WObj:=Workobject_1;
        MoveL point_548_clearance,v500,fine,GS25_ParallelGripper\WObj:=Workobject_1;
        MoveL point_548_contact,v500,fine,GS25_ParallelGripper\WObj:=Workobject_1;
        MoveL point_549_contact,v500,fine,GS25_ParallelGripper\WObj:=Workobject_1;
        MoveL point_549_clearance,v500,fine,GS25_ParallelGripper\WObj:=Workobject_1;
        MoveL point_550_clearance,v500,fine,GS25_ParallelGripper\WObj:=Workobject_1;
        MoveL point_550_contact,v500,fine,GS25_ParallelGripper\WObj:=Workobject_1;
        MoveL point_551_contact,v500,fine,GS25_ParallelGripper\WObj:=Workobject_1;
        MoveL point_551_clearance,v500,fine,GS25_ParallelGripper\WObj:=Workobject_1;
        MoveL point_552_clearance,v500,fine,GS25_ParallelGripper\WObj:=Workobject_1;
        MoveL point_552_contact,v500,fine,GS25_ParallelGripper\WObj:=Workobject_1;
        MoveL point_553_contact,v500,fine,GS25_ParallelGripper\WObj:=Workobject_1;
        MoveL point_553_clearance,v500,fine,GS25_ParallelGripper\WObj:=Workobject_1;
        MoveL point_554_clearance,v500,fine,GS25_ParallelGripper\WObj:=Workobject_1;
        MoveL point_554_contact,v500,fine,GS25_ParallelGripper\WObj:=Workobject_1;
        MoveL point_555_contact,v500,fine,GS25_ParallelGripper\WObj:=Workobject_1;
        MoveL point_555_clearance,v500,fine,GS25_ParallelGripper\WObj:=Workobject_1;
        MoveL point_556_clearance,v500,fine,GS25_ParallelGripper\WObj:=Workobject_1;
        MoveL point_556_contact,v500,fine,GS25_ParallelGripper\WObj:=Workobject_1;
        MoveL point_557_contact,v500,fine,GS25_ParallelGripper\WObj:=Workobject_1;
        MoveL point_557_clearance,v500,fine,GS25_ParallelGripper\WObj:=Workobject_1;
        MoveL point_558_clearance,v500,fine,GS25_ParallelGripper\WObj:=Workobject_1;
        MoveL point_558_contact,v500,fine,GS25_ParallelGripper\WObj:=Workobject_1;
        MoveL point_559_contact,v500,fine,GS25_ParallelGripper\WObj:=Workobject_1;
        MoveL point_559_clearance,v500,fine,GS25_ParallelGripper\WObj:=Workobject_1;
        MoveL point_560_clearance,v500,fine,GS25_ParallelGripper\WObj:=Workobject_1;
        MoveL point_560_contact,v500,fine,GS25_ParallelGripper\WObj:=Workobject_1;
        MoveL point_561_contact,v500,fine,GS25_ParallelGripper\WObj:=Workobject_1;
        MoveL point_561_clearance,v500,fine,GS25_ParallelGripper\WObj:=Workobject_1;
        MoveL point_562_clearance,v500,fine,GS25_ParallelGripper\WObj:=Workobject_1;
        MoveL point_562_contact,v500,fine,GS25_ParallelGripper\WObj:=Workobject_1;
        MoveL point_563_contact,v500,fine,GS25_ParallelGripper\WObj:=Workobject_1;
        MoveL point_563_clearance,v500,fine,GS25_ParallelGripper\WObj:=Workobject_1;
        MoveL point_564_clearance,v500,fine,GS25_ParallelGripper\WObj:=Workobject_1;
        MoveL point_564_contact,v500,fine,GS25_ParallelGripper\WObj:=Workobject_1;
        MoveL point_565_contact,v500,fine,GS25_ParallelGripper\WObj:=Workobject_1;
        MoveL point_565_clearance,v500,fine,GS25_ParallelGripper\WObj:=Workobject_1;
        MoveL point_566_clearance,v500,fine,GS25_ParallelGripper\WObj:=Workobject_1;
        MoveL point_566_contact,v500,fine,GS25_ParallelGripper\WObj:=Workobject_1;
        MoveL point_567_contact,v500,fine,GS25_ParallelGripper\WObj:=Workobject_1;
        MoveL point_567_clearance,v500,fine,GS25_ParallelGripper\WObj:=Workobject_1;
        MoveL point_568_clearance,v500,fine,GS25_ParallelGripper\WObj:=Workobject_1;
        MoveL point_568_contact,v500,fine,GS25_ParallelGripper\WObj:=Workobject_1;
        MoveL point_569_contact,v500,fine,GS25_ParallelGripper\WObj:=Workobject_1;
        MoveL point_569_clearance,v500,fine,GS25_ParallelGripper\WObj:=Workobject_1;
        MoveL point_570_clearance,v500,fine,GS25_ParallelGripper\WObj:=Workobject_1;
        MoveL point_570_contact,v500,fine,GS25_ParallelGripper\WObj:=Workobject_1;
        MoveL point_571_contact,v500,fine,GS25_ParallelGripper\WObj:=Workobject_1;
        MoveL point_571_clearance,v500,fine,GS25_ParallelGripper\WObj:=Workobject_1;
        MoveL point_572_clearance,v500,fine,GS25_ParallelGripper\WObj:=Workobject_1;
        MoveL point_572_contact,v500,fine,GS25_ParallelGripper\WObj:=Workobject_1;
        MoveL point_573_contact,v500,fine,GS25_ParallelGripper\WObj:=Workobject_1;
        MoveL point_573_clearance,v500,fine,GS25_ParallelGripper\WObj:=Workobject_1;
        MoveL point_574_clearance,v500,fine,GS25_ParallelGripper\WObj:=Workobject_1;
        MoveL point_574_contact,v500,fine,GS25_ParallelGripper\WObj:=Workobject_1;
        MoveL point_575_contact,v500,fine,GS25_ParallelGripper\WObj:=Workobject_1;
        MoveL point_575_clearance,v500,fine,GS25_ParallelGripper\WObj:=Workobject_1;
        MoveL point_576_clearance,v500,fine,GS25_ParallelGripper\WObj:=Workobject_1;
        MoveL point_576_contact,v500,fine,GS25_ParallelGripper\WObj:=Workobject_1;
        MoveL point_577_contact,v500,fine,GS25_ParallelGripper\WObj:=Workobject_1;
        MoveL point_577_clearance,v500,fine,GS25_ParallelGripper\WObj:=Workobject_1;
        MoveL point_578_clearance,v500,fine,GS25_ParallelGripper\WObj:=Workobject_1;
        MoveL point_578_contact,v500,fine,GS25_ParallelGripper\WObj:=Workobject_1;
        MoveL point_579_contact,v500,fine,GS25_ParallelGripper\WObj:=Workobject_1;
        MoveL point_579_clearance,v500,fine,GS25_ParallelGripper\WObj:=Workobject_1;
        MoveL point_580_clearance,v500,fine,GS25_ParallelGripper\WObj:=Workobject_1;
        MoveL point_580_contact,v500,fine,GS25_ParallelGripper\WObj:=Workobject_1;
        MoveL point_581_contact,v500,fine,GS25_ParallelGripper\WObj:=Workobject_1;
        MoveL point_581_clearance,v500,fine,GS25_ParallelGripper\WObj:=Workobject_1;
        MoveL point_582_clearance,v500,fine,GS25_ParallelGripper\WObj:=Workobject_1;
        MoveL point_582_contact,v500,fine,GS25_ParallelGripper\WObj:=Workobject_1;
        MoveL point_583_contact,v500,fine,GS25_ParallelGripper\WObj:=Workobject_1;
        MoveL point_583_clearance,v500,fine,GS25_ParallelGripper\WObj:=Workobject_1;
        MoveL point_584_clearance,v500,fine,GS25_ParallelGripper\WObj:=Workobject_1;
        MoveL point_584_contact,v500,fine,GS25_ParallelGripper\WObj:=Workobject_1;
        MoveL point_585_contact,v500,fine,GS25_ParallelGripper\WObj:=Workobject_1;
        MoveL point_585_clearance,v500,fine,GS25_ParallelGripper\WObj:=Workobject_1;
        MoveL point_586_clearance,v500,fine,GS25_ParallelGripper\WObj:=Workobject_1;
        MoveL point_586_contact,v500,fine,GS25_ParallelGripper\WObj:=Workobject_1;
        MoveL point_587_contact,v500,fine,GS25_ParallelGripper\WObj:=Workobject_1;
        MoveL point_587_clearance,v500,fine,GS25_ParallelGripper\WObj:=Workobject_1;
        MoveL point_588_clearance,v500,fine,GS25_ParallelGripper\WObj:=Workobject_1;
        MoveL point_588_contact,v500,fine,GS25_ParallelGripper\WObj:=Workobject_1;
        MoveL point_589_contact,v500,fine,GS25_ParallelGripper\WObj:=Workobject_1;
        MoveL point_589_clearance,v500,fine,GS25_ParallelGripper\WObj:=Workobject_1;
        MoveL point_590_clearance,v500,fine,GS25_ParallelGripper\WObj:=Workobject_1;
        MoveL point_590_contact,v500,fine,GS25_ParallelGripper\WObj:=Workobject_1;
        MoveL point_591_contact,v500,fine,GS25_ParallelGripper\WObj:=Workobject_1;
        MoveL point_591_clearance,v500,fine,GS25_ParallelGripper\WObj:=Workobject_1;
        MoveL point_592_clearance,v500,fine,GS25_ParallelGripper\WObj:=Workobject_1;
        MoveL point_592_contact,v500,fine,GS25_ParallelGripper\WObj:=Workobject_1;
        MoveL point_593_contact,v500,fine,GS25_ParallelGripper\WObj:=Workobject_1;
        MoveL point_593_clearance,v500,fine,GS25_ParallelGripper\WObj:=Workobject_1;
        MoveL point_594_clearance,v500,fine,GS25_ParallelGripper\WObj:=Workobject_1;
        MoveL point_594_contact,v500,fine,GS25_ParallelGripper\WObj:=Workobject_1;
        MoveL point_595_contact,v500,fine,GS25_ParallelGripper\WObj:=Workobject_1;
        MoveL point_595_clearance,v500,fine,GS25_ParallelGripper\WObj:=Workobject_1;
